    movel(p[x_c + 0.072285, y_c + -0.106434, z_c, rx, ry, rz], a, v)
    movel(p[x_c + 0.072329, y_c + -0.106475, z_c, rx, ry, rz], a, v)
    movel(p[x_c + 0.072376, y_c + -0.106518, z_c, rx, ry, rz], a, v)
    movel(p[x_c + 0.072426, y_c + -0.106564, z_c, rx, ry, rz], a, v)
    movel(p[x_c + 0.072479, y_c + -0.106612, z_c, rx, ry, rz], a, v)
    movel(p[x_c + 0.072535, y_c + -0.106663, z_c, rx, ry, rz], a, v)
    movel(p[x_c + 0.072593, y_c + -0.106716, z_c, rx, ry, rz], a, v)
    movel(p[x_c + 0.072654, y_c + -0.106772, z_c, rx, ry, rz], a, v)
    movel(p[x_c + 0.072718, y_c + -0.106830, z_c, rx, ry, rz], a, v)
    movel(p[x_c + 0.072785, y_c + -0.106890, z_c, rx, ry, rz], a, v)
    movel(p[x_c + 0.072855, y_c + -0.106954, z_c, rx, ry, rz], a, v)
    movel(p[x_c + 0.072855, y_c + -0.106954, z_c, rx, ry, rz], a, v)
    movel(p[x_c + 0.072959, y_c + -0.107049, z_c, rx, ry, rz], a, v)
    movel(p[x_c + 0.073072, y_c + -0.107153, z_c, rx, ry, rz], a, v)
    movel(p[x_c + 0.073193, y_c + -0.107267, z_c, rx, ry, rz], a, v)
    movel(p[x_c + 0.073322, y_c + -0.107389, z_c, rx, ry, rz], a, v)
    movel(p[x_c + 0.073459, y_c + -0.107519, z_c, rx, ry, rz], a, v)
    movel(p[x_c + 0.073603, y_c + -0.107657, z_c, rx, ry, rz], a, v)
    movel(p[x_c + 0.073754, y_c + -0.107802, z_c, rx, ry, rz], a, v)
    movel(p[x_c + 0.073910, y_c + -0.107953, z_c, rx, ry, rz], a, v)
    movel(p[x_c + 0.074072, y_c + -0.108111, z_c, rx, ry, rz], a, v)
    movel(p[x_c + 0.074240, y_c + -0.108275, z_c, rx, ry, rz], a, v)
    movel(p[x_c + 0.074412, y_c + -0.108443, z_c, rx, ry, rz], a, v)
    movel(p[x_c + 0.074589, y_c + -0.108617, z_c, rx, ry, rz], a, v)
    movel(p[x_c + 0.074769, y_c + -0.108795, z_c, rx, ry, rz], a, v)
    movel(p[x_c + 0.074953, y_c + -0.108977, z_c, rx, ry, rz], a, v)
    movel(p[x_c + 0.075139, y_c + -0.109162, z_c, rx, ry, rz], a, v)
    movel(p[x_c + 0.075329, y_c + -0.109350, z_c, rx, ry, rz], a, v)
    movel(p[x_c + 0.075520, y_c + -0.109541, z_c, rx, ry, rz], a, v)
    movel(p[x_c + 0.075712, y_c + -0.109734, z_c, rx, ry, rz], a, v)
    movel(p[x_c + 0.075906, y_c + -0.109928, z_c, rx, ry, rz], a, v)
    movel(p[x_c + 0.076100, y_c + -0.110123, z_c, rx, ry, rz], a, v)
    movel(p[x_c + 0.076295, y_c + -0.110319, z_c, rx, ry, rz], a, v)
    movel(p[x_c + 0.076489, y_c + -0.110515, z_c, rx, ry, rz], a, v)
    movel(p[x_c + 0.076683, y_c + -0.110711, z_c, rx, ry, rz], a, v)
    movel(p[x_c + 0.076875, y_c + -0.110906, z_c, rx, ry, rz], a, v)
    movel(p[x_c + 0.077065, y_c + -0.111099, z_c, rx, ry, rz], a, v)
    movel(p[x_c + 0.077254, y_c + -0.111291, z_c, rx, ry, rz], a, v)
    movel(p[x_c + 0.077440, y_c + -0.111481, z_c, rx, ry, rz], a, v)
    movel(p[x_c + 0.077622, y_c + -0.111668, z_c, rx, ry, rz], a, v)
    movel(p[x_c + 0.077802, y_c + -0.111852, z_c, rx, ry, rz], a, v)
    movel(p[x_c + 0.077977, y_c + -0.112032, z_c, rx, ry, rz], a, v)
    movel(p[x_c + 0.078148, y_c + -0.112209, z_c, rx, ry, rz], a, v)
    movel(p[x_c + 0.078314, y_c + -0.112380, z_c, rx, ry, rz], a, v)
    movel(p[x_c + 0.078474, y_c + -0.112547, z_c, rx, ry, rz], a, v)
    movel(p[x_c + 0.078629, y_c + -0.112708, z_c, rx, ry, rz], a, v)
    movel(p[x_c + 0.078778, y_c + -0.112864, z_c, rx, ry, rz], a, v)
    movel(p[x_c + 0.078919, y_c + -0.113013, z_c, rx, ry, rz], a, v)
    movel(p[x_c + 0.079054, y_c + -0.113155, z_c, rx, ry, rz], a, v)
    movel(p[x_c + 0.079181, y_c + -0.113290, z_c, rx, ry, rz], a, v)
    movel(p[x_c + 0.079300, y_c + -0.113417, z_c, rx, ry, rz], a, v)
    movel(p[x_c + 0.079410, y_c + -0.113535, z_c, rx, ry, rz], a, v)
    movel(p[x_c + 0.079511, y_c + -0.113645, z_c, rx, ry, rz], a, v)
    movel(p[x_c + 0.079603, y_c + -0.113746, z_c, rx, ry, rz], a, v)
    movel(p[x_c + 0.079685, y_c + -0.113837, z_c, rx, ry, rz], a, v)
    movel(p[x_c + 0.079756, y_c + -0.113918, z_c, rx, ry, rz], a, v)
    movel(p[x_c + 0.079817, y_c + -0.113989, z_c, rx, ry, rz], a, v)
    movel(p[x_c + 0.079866, y_c + -0.114048, z_c, rx, ry, rz], a, v)
    movel(p[x_c + 0.079904, y_c + -0.114096, z_c, rx, ry, rz], a, v)
    movel(p[x_c + 0.079929, y_c + -0.114132, z_c, rx, ry, rz], a, v)
    movel(p[x_c + 0.079941, y_c + -0.114155, z_c, rx, ry, rz], a, v)
    movel(p[x_c + 0.079941, y_c + -0.114155, z_c, rx, ry, rz], a, v)
    movel(p[x_c + 0.079943, y_c + -0.114162, z_c, rx, ry, rz], a, v)
    movel(p[x_c + 0.079943, y_c + -0.114167, z_c, rx, ry, rz], a, v)
    movel(p[x_c + 0.079941, y_c + -0.114171, z_c, rx, ry, rz], a, v)
    movel(p[x_c + 0.079937, y_c + -0.114173, z_c, rx, ry, rz], a, v)
    movel(p[x_c + 0.079932, y_c + -0.114175, z_c, rx, ry, rz], a, v)
    movel(p[x_c + 0.079924, y_c + -0.114175, z_c, rx, ry, rz], a, v)
    movel(p[x_c + 0.079916, y_c + -0.114173, z_c, rx, ry, rz], a, v)
    movel(p[x_c + 0.079905, y_c + -0.114171, z_c, rx, ry, rz], a, v)
    movel(p[x_c + 0.079892, y_c + -0.114167, z_c, rx, ry, rz], a, v)
    movel(p[x_c + 0.079878, y_c + -0.114162, z_c, rx, ry, rz], a, v)
    movel(p[x_c + 0.079863, y_c + -0.114155, z_c, rx, ry, rz], a, v)
    movel(p[x_c + 0.079846, y_c + -0.114148, z_c, rx, ry, rz], a, v)
    movel(p[x_c + 0.079827, y_c + -0.114139, z_c, rx, ry, rz], a, v)
    movel(p[x_c + 0.079807, y_c + -0.114129, z_c, rx, ry, rz], a, v)
    movel(p[x_c + 0.079785, y_c + -0.114119, z_c, rx, ry, rz], a, v)
    movel(p[x_c + 0.079762, y_c + -0.114106, z_c, rx, ry, rz], a, v)
    movel(p[x_c + 0.079737, y_c + -0.114093, z_c, rx, ry, rz], a, v)
    movel(p[x_c + 0.079711, y_c + -0.114079, z_c, rx, ry, rz], a, v)
    movel(p[x_c + 0.079684, y_c + -0.114064, z_c, rx, ry, rz], a, v)
    movel(p[x_c + 0.079655, y_c + -0.114047, z_c, rx, ry, rz], a, v)
    movel(p[x_c + 0.079625, y_c + -0.114030, z_c, rx, ry, rz], a, v)
    movel(p[x_c + 0.079593, y_c + -0.114012, z_c, rx, ry, rz], a, v)
    movel(p[x_c + 0.079561, y_c + -0.113992, z_c, rx, ry, rz], a, v)
    movel(p[x_c + 0.079527, y_c + -0.113972, z_c, rx, ry, rz], a, v)
    movel(p[x_c + 0.079492, y_c + -0.113950, z_c, rx, ry, rz], a, v)
    movel(p[x_c + 0.079455, y_c + -0.113928, z_c, rx, ry, rz], a, v)
    movel(p[x_c + 0.079418, y_c + -0.113905, z_c, rx, ry, rz], a, v)
    movel(p[x_c + 0.079379, y_c + -0.113881, z_c, rx, ry, rz], a, v)
    movel(p[x_c + 0.079340, y_c + -0.113856, z_c, rx, ry, rz], a, v)
    movel(p[x_c + 0.079299, y_c + -0.113830, z_c, rx, ry, rz], a, v)
    movel(p[x_c + 0.079257, y_c + -0.113803, z_c, rx, ry, rz], a, v)
    movel(p[x_c + 0.079214, y_c + -0.113775, z_c, rx, ry, rz], a, v)
    movel(p[x_c + 0.079171, y_c + -0.113747, z_c, rx, ry, rz], a, v)
    movel(p[x_c + 0.079126, y_c + -0.113718, z_c, rx, ry, rz], a, v)
    movel(p[x_c + 0.079080, y_c + -0.113688, z_c, rx, ry, rz], a, v)
    movel(p[x_c + 0.079034, y_c + -0.113657, z_c, rx, ry, rz], a, v)
    movel(p[x_c + 0.078987, y_c + -0.113625, z_c, rx, ry, rz], a, v)
    movel(p[x_c + 0.078938, y_c + -0.113593, z_c, rx, ry, rz], a, v)
    movel(p[x_c + 0.078889, y_c + -0.113560, z_c, rx, ry, rz], a, v)
    movel(p[x_c + 0.078840, y_c + -0.113526, z_c, rx, ry, rz], a, v)
    movel(p[x_c + 0.078789, y_c + -0.113492, z_c, rx, ry, rz], a, v)
    movel(p[x_c + 0.078738, y_c + -0.113457, z_c, rx, ry, rz], a, v)
    movel(p[x_c + 0.078686, y_c + -0.113421, z_c, rx, ry, rz], a, v)
    movel(p[x_c + 0.078633, y_c + -0.113384, z_c, rx, ry, rz], a, v)
    movel(p[x_c + 0.078580, y_c + -0.113347, z_c, rx, ry, rz], a, v)
    movel(p[x_c + 0.078526, y_c + -0.113310, z_c, rx, ry, rz], a, v)
    movel(p[x_c + 0.078472, y_c + -0.113272, z_c, rx, ry, rz], a, v)
    movel(p[x_c + 0.078417, y_c + -0.113233, z_c, rx, ry, rz], a, v)
    movel(p[x_c + 0.078361, y_c + -0.113193, z_c, rx, ry, rz], a, v)
    movel(p[x_c + 0.078361, y_c + -0.113193, z_c, rx, ry, rz], a, v)
    movel(p[x_c + 0.078071, y_c + -0.112987, z_c, rx, ry, rz], a, v)
    movel(p[x_c + 0.077789, y_c + -0.112787, z_c, rx, ry, rz], a, v)
    movel(p[x_c + 0.077513, y_c + -0.112592, z_c, rx, ry, rz], a, v)
    movel(p[x_c + 0.077245, y_c + -0.112401, z_c, rx, ry, rz], a, v)
    movel(p[x_c + 0.076983, y_c + -0.112216, z_c, rx, ry, rz], a, v)
    movel(p[x_c + 0.076728, y_c + -0.112036, z_c, rx, ry, rz], a, v)
    movel(p[x_c + 0.076480, y_c + -0.111861, z_c, rx, ry, rz], a, v)
    movel(p[x_c + 0.076238, y_c + -0.111690, z_c, rx, ry, rz], a, v)
    movel(p[x_c + 0.076002, y_c + -0.111524, z_c, rx, ry, rz], a, v)
    movel(p[x_c + 0.075773, y_c + -0.111363, z_c, rx, ry, rz], a, v)
    movel(p[x_c + 0.075549, y_c + -0.111206, z_c, rx, ry, rz], a, v)
    movel(p[x_c + 0.075331, y_c + -0.111054, z_c, rx, ry, rz], a, v)
    movel(p[x_c + 0.075119, y_c + -0.110905, z_c, rx, ry, rz], a, v)
    movel(p[x_c + 0.074913, y_c + -0.110761, z_c, rx, ry, rz], a, v)
    movel(p[x_c + 0.074711, y_c + -0.110621, z_c, rx, ry, rz], a, v)
    movel(p[x_c + 0.074515, y_c + -0.110485, z_c, rx, ry, rz], a, v)
    movel(p[x_c + 0.074324, y_c + -0.110353, z_c, rx, ry, rz], a, v)
    movel(p[x_c + 0.074138, y_c + -0.110224, z_c, rx, ry, rz], a, v)
    movel(p[x_c + 0.073957, y_c + -0.110099, z_c, rx, ry, rz], a, v)
    movel(p[x_c + 0.073780, y_c + -0.109978, z_c, rx, ry, rz], a, v)
    movel(p[x_c + 0.073608, y_c + -0.109860, z_c, rx, ry, rz], a, v)
    movel(p[x_c + 0.073440, y_c + -0.109745, z_c, rx, ry, rz], a, v)
    movel(p[x_c + 0.073276, y_c + -0.109634, z_c, rx, ry, rz], a, v)
    movel(p[x_c + 0.073117, y_c + -0.109526, z_c, rx, ry, rz], a, v)
    movel(p[x_c + 0.072961, y_c + -0.109420, z_c, rx, ry, rz], a, v)
    movel(p[x_c + 0.072809, y_c + -0.109318, z_c, rx, ry, rz], a, v)
    movel(p[x_c + 0.072660, y_c + -0.109219, z_c, rx, ry, rz], a, v)
    movel(p[x_c + 0.072515, y_c + -0.109122, z_c, rx, ry, rz], a, v)
    movel(p[x_c + 0.072373, y_c + -0.109028, z_c, rx, ry, rz], a, v)
    movel(p[x_c + 0.072234, y_c + -0.108936, z_c, rx, ry, rz], a, v)
    movel(p[x_c + 0.072098, y_c + -0.108847, z_c, rx, ry, rz], a, v)
    movel(p[x_c + 0.071965, y_c + -0.108760, z_c, rx, ry, rz], a, v)
    movel(p[x_c + 0.071834, y_c + -0.108675, z_c, rx, ry, rz], a, v)
    movel(p[x_c + 0.071706, y_c + -0.108593, z_c, rx, ry, rz], a, v)
    movel(p[x_c + 0.071581, y_c + -0.108512, z_c, rx, ry, rz], a, v)
    movel(p[x_c + 0.071457, y_c + -0.108433, z_c, rx, ry, rz], a, v)
    movel(p[x_c + 0.071336, y_c + -0.108357, z_c, rx, ry, rz], a, v)
    movel(p[x_c + 0.071216, y_c + -0.108281, z_c, rx, ry, rz], a, v)
    movel(p[x_c + 0.071099, y_c + -0.108208, z_c, rx, ry, rz], a, v)
    movel(p[x_c + 0.070983, y_c + -0.108136, z_c, rx, ry, rz], a, v)
    movel(p[x_c + 0.070868, y_c + -0.108065, z_c, rx, ry, rz], a, v)
    movel(p[x_c + 0.070755, y_c + -0.107996, z_c, rx, ry, rz], a, v)
    movel(p[x_c + 0.070642, y_c + -0.107928, z_c, rx, ry, rz], a, v)
    movel(p[x_c + 0.070531, y_c + -0.107861, z_c, rx, ry, rz], a, v)
    movel(p[x_c + 0.070421, y_c + -0.107795, z_c, rx, ry, rz], a, v)
    movel(p[x_c + 0.070311, y_c + -0.107729, z_c, rx, ry, rz], a, v)
    movel(p[x_c + 0.070202, y_c + -0.107665, z_c, rx, ry, rz], a, v)
    movel(p[x_c + 0.070093, y_c + -0.107601, z_c, rx, ry, rz], a, v)
    movel(p[x_c + 0.069984, y_c + -0.107538, z_c, rx, ry, rz], a, v)
    movel(p[x_c + 0.069984, y_c + -0.107538, z_c, rx, ry, rz], a, v)
    movel(p[x_c + 0.069919, y_c + -0.107500, z_c, rx, ry, rz], a, v)
    movel(p[x_c + 0.069853, y_c + -0.107462, z_c, rx, ry, rz], a, v)
    movel(p[x_c + 0.069787, y_c + -0.107423, z_c, rx, ry, rz], a, v)
    movel(p[x_c + 0.069721, y_c + -0.107385, z_c, rx, ry, rz], a, v)
    movel(p[x_c + 0.069654, y_c + -0.107346, z_c, rx, ry, rz], a, v)
    movel(p[x_c + 0.069588, y_c + -0.107308, z_c, rx, ry, rz], a, v)
    movel(p[x_c + 0.069522, y_c + -0.107269, z_c, rx, ry, rz], a, v)
    movel(p[x_c + 0.069456, y_c + -0.107230, z_c, rx, ry, rz], a, v)
    movel(p[x_c + 0.069391, y_c + -0.107192, z_c, rx, ry, rz], a, v)
    movel(p[x_c + 0.069325, y_c + -0.107153, z_c, rx, ry, rz], a, v)
    movel(p[x_c + 0.069260, y_c + -0.107115, z_c, rx, ry, rz], a, v)
    movel(p[x_c + 0.069195, y_c + -0.107077, z_c, rx, ry, rz], a, v)
    movel(p[x_c + 0.069130, y_c + -0.107039, z_c, rx, ry, rz], a, v)
    movel(p[x_c + 0.069066, y_c + -0.107001, z_c, rx, ry, rz], a, v)
    movel(p[x_c + 0.069002, y_c + -0.106963, z_c, rx, ry, rz], a, v)
    movel(p[x_c + 0.068939, y_c + -0.106926, z_c, rx, ry, rz], a, v)
    movel(p[x_c + 0.068876, y_c + -0.106889, z_c, rx, ry, rz], a, v)
    movel(p[x_c + 0.068814, y_c + -0.106852, z_c, rx, ry, rz], a, v)
    movel(p[x_c + 0.068752, y_c + -0.106815, z_c, rx, ry, rz], a, v)
    movel(p[x_c + 0.068691, y_c + -0.106779, z_c, rx, ry, rz], a, v)
    movel(p[x_c + 0.068631, y_c + -0.106743, z_c, rx, ry, rz], a, v)
    movel(p[x_c + 0.068572, y_c + -0.106708, z_c, rx, ry, rz], a, v)
    movel(p[x_c + 0.068513, y_c + -0.106673, z_c, rx, ry, rz], a, v)
    movel(p[x_c + 0.068455, y_c + -0.106639, z_c, rx, ry, rz], a, v)
    movel(p[x_c + 0.068398, y_c + -0.106605, z_c, rx, ry, rz], a, v)
    movel(p[x_c + 0.068342, y_c + -0.106571, z_c, rx, ry, rz], a, v)
    movel(p[x_c + 0.068287, y_c + -0.106538, z_c, rx, ry, rz], a, v)
    movel(p[x_c + 0.068233, y_c + -0.106506, z_c, rx, ry, rz], a, v)
    movel(p[x_c + 0.068181, y_c + -0.106474, z_c, rx, ry, rz], a, v)
    movel(p[x_c + 0.068129, y_c + -0.106443, z_c, rx, ry, rz], a, v)
    movel(p[x_c + 0.068078, y_c + -0.106412, z_c, rx, ry, rz], a, v)
    movel(p[x_c + 0.068029, y_c + -0.106382, z_c, rx, ry, rz], a, v)
    movel(p[x_c + 0.067981, y_c + -0.106353, z_c, rx, ry, rz], a, v)
    movel(p[x_c + 0.067934, y_c + -0.106325, z_c, rx, ry, rz], a, v)
    movel(p[x_c + 0.067889, y_c + -0.106297, z_c, rx, ry, rz], a, v)
    movel(p[x_c + 0.067844, y_c + -0.106270, z_c, rx, ry, rz], a, v)
    movel(p[x_c + 0.067802, y_c + -0.106244, z_c, rx, ry, rz], a, v)
    movel(p[x_c + 0.067761, y_c + -0.106219, z_c, rx, ry, rz], a, v)
    movel(p[x_c + 0.067721, y_c + -0.106195, z_c, rx, ry, rz], a, v)
    movel(p[x_c + 0.067683, y_c + -0.106171, z_c, rx, ry, rz], a, v)
    movel(p[x_c + 0.067647, y_c + -0.106149, z_c, rx, ry, rz], a, v)
    movel(p[x_c + 0.067612, y_c + -0.106127, z_c, rx, ry, rz], a, v)
    movel(p[x_c + 0.067579, y_c + -0.106107, z_c, rx, ry, rz], a, v)
    movel(p[x_c + 0.067548, y_c + -0.106087, z_c, rx, ry, rz], a, v)
    movel(p[x_c + 0.067519, y_c + -0.106069, z_c, rx, ry, rz], a, v)
    movel(p[x_c + 0.067491, y_c + -0.106051, z_c, rx, ry, rz], a, v)
    movel(p[x_c + 0.067466, y_c + -0.106035, z_c, rx, ry, rz], a, v)
    movel(p[x_c + 0.067442, y_c + -0.106020, z_c, rx, ry, rz], a, v)
    movel(p[x_c + 0.067420, y_c + -0.106006, z_c, rx, ry, rz], a, v)
    movel(p[x_c + 0.067420, y_c + -0.106006, z_c, rx, ry, rz], a, v)
    movel(p[x_c + 0.067361, y_c + -0.105967, z_c, rx, ry, rz], a, v)
    movel(p[x_c + 0.067304, y_c + -0.105930, z_c, rx, ry, rz], a, v)
    movel(p[x_c + 0.067251, y_c + -0.105897, z_c, rx, ry, rz], a, v)
    movel(p[x_c + 0.067201, y_c + -0.105865, z_c, rx, ry, rz], a, v)
    movel(p[x_c + 0.067154, y_c + -0.105837, z_c, rx, ry, rz], a, v)
    movel(p[x_c + 0.067110, y_c + -0.105810, z_c, rx, ry, rz], a, v)
    movel(p[x_c + 0.067070, y_c + -0.105787, z_c, rx, ry, rz], a, v)
    movel(p[x_c + 0.067032, y_c + -0.105765, z_c, rx, ry, rz], a, v)
    movel(p[x_c + 0.066998, y_c + -0.105746, z_c, rx, ry, rz], a, v)
    movel(p[x_c + 0.066966, y_c + -0.105729, z_c, rx, ry, rz], a, v)
    movel(p[x_c + 0.066938, y_c + -0.105715, z_c, rx, ry, rz], a, v)
    movel(p[x_c + 0.066912, y_c + -0.105703, z_c, rx, ry, rz], a, v)
    movel(p[x_c + 0.066890, y_c + -0.105693, z_c, rx, ry, rz], a, v)
    movel(p[x_c + 0.066870, y_c + -0.105685, z_c, rx, ry, rz], a, v)
    movel(p[x_c + 0.066853, y_c + -0.105679, z_c, rx, ry, rz], a, v)
    movel(p[x_c + 0.066839, y_c + -0.105676, z_c, rx, ry, rz], a, v)
    movel(p[x_c + 0.066828, y_c + -0.105674, z_c, rx, ry, rz], a, v)
    movel(p[x_c + 0.066820, y_c + -0.105675, z_c, rx, ry, rz], a, v)
    movel(p[x_c + 0.066815, y_c + -0.105677, z_c, rx, ry, rz], a, v)
    movel(p[x_c + 0.066812, y_c + -0.105682, z_c, rx, ry, rz], a, v)
    movel(p[x_c + 0.066812, y_c + -0.105689, z_c, rx, ry, rz], a, v)
    movel(p[x_c + 0.066815, y_c + -0.105697, z_c, rx, ry, rz], a, v)
    movel(p[x_c + 0.066821, y_c + -0.105708, z_c, rx, ry, rz], a, v)
    movel(p[x_c + 0.066829, y_c + -0.105720, z_c, rx, ry, rz], a, v)
    movel(p[x_c + 0.066840, y_c + -0.105734, z_c, rx, ry, rz], a, v)
    movel(p[x_c + 0.066853, y_c + -0.105750, z_c, rx, ry, rz], a, v)
    movel(p[x_c + 0.066869, y_c + -0.105768, z_c, rx, ry, rz], a, v)
    movel(p[x_c + 0.066888, y_c + -0.105787, z_c, rx, ry, rz], a, v)
    movel(p[x_c + 0.066909, y_c + -0.105808, z_c, rx, ry, rz], a, v)
    movel(p[x_c + 0.066933, y_c + -0.105831, z_c, rx, ry, rz], a, v)
    movel(p[x_c + 0.066959, y_c + -0.105855, z_c, rx, ry, rz], a, v)
    movel(p[x_c + 0.066988, y_c + -0.105881, z_c, rx, ry, rz], a, v)
    movel(p[x_c + 0.067019, y_c + -0.105909, z_c, rx, ry, rz], a, v)
    movel(p[x_c + 0.067053, y_c + -0.105938, z_c, rx, ry, rz], a, v)
    movel(p[x_c + 0.067089, y_c + -0.105969, z_c, rx, ry, rz], a, v)
    movel(p[x_c + 0.067127, y_c + -0.106001, z_c, rx, ry, rz], a, v)
    movel(p[x_c + 0.067168, y_c + -0.106034, z_c, rx, ry, rz], a, v)
    movel(p[x_c + 0.067211, y_c + -0.106069, z_c, rx, ry, rz], a, v)
    movel(p[x_c + 0.067256, y_c + -0.106106, z_c, rx, ry, rz], a, v)
    movel(p[x_c + 0.067304, y_c + -0.106143, z_c, rx, ry, rz], a, v)
    movel(p[x_c + 0.067353, y_c + -0.106182, z_c, rx, ry, rz], a, v)
    movel(p[x_c + 0.067405, y_c + -0.106223, z_c, rx, ry, rz], a, v)
    movel(p[x_c + 0.067460, y_c + -0.106264, z_c, rx, ry, rz], a, v)
    movel(p[x_c + 0.067516, y_c + -0.106307, z_c, rx, ry, rz], a, v)
    movel(p[x_c + 0.067575, y_c + -0.106351, z_c, rx, ry, rz], a, v)
    movel(p[x_c + 0.067635, y_c + -0.106396, z_c, rx, ry, rz], a, v)
    movel(p[x_c + 0.067698, y_c + -0.106442, z_c, rx, ry, rz], a, v)
    movel(p[x_c + 0.067763, y_c + -0.106489, z_c, rx, ry, rz], a, v)
    movel(p[x_c + 0.067830, y_c + -0.106537, z_c, rx, ry, rz], a, v)
    movel(p[x_c + 0.067830, y_c + -0.106537, z_c, rx, ry, rz], a, v)
    movel(p[x_c + 0.067865, y_c + -0.106563, z_c, rx, ry, rz], a, v)
    movel(p[x_c + 0.067903, y_c + -0.106591, z_c, rx, ry, rz], a, v)
    movel(p[x_c + 0.067944, y_c + -0.106620, z_c, rx, ry, rz], a, v)
    movel(p[x_c + 0.067986, y_c + -0.106652, z_c, rx, ry, rz], a, v)
    movel(p[x_c + 0.068031, y_c + -0.106685, z_c, rx, ry, rz], a, v)
    movel(p[x_c + 0.068077, y_c + -0.106721, z_c, rx, ry, rz], a, v)
    movel(p[x_c + 0.068126, y_c + -0.106758, z_c, rx, ry, rz], a, v)
    movel(p[x_c + 0.068177, y_c + -0.106797, z_c, rx, ry, rz], a, v)
    movel(p[x_c + 0.068229, y_c + -0.106837, z_c, rx, ry, rz], a, v)
    movel(p[x_c + 0.068284, y_c + -0.106879, z_c, rx, ry, rz], a, v)
    movel(p[x_c + 0.068340, y_c + -0.106922, z_c, rx, ry, rz], a, v)
    movel(p[x_c + 0.068398, y_c + -0.106968, z_c, rx, ry, rz], a, v)
    movel(p[x_c + 0.068458, y_c + -0.107014, z_c, rx, ry, rz], a, v)
    movel(p[x_c + 0.068519, y_c + -0.107062, z_c, rx, ry, rz], a, v)
    movel(p[x_c + 0.068582, y_c + -0.107111, z_c, rx, ry, rz], a, v)
    movel(p[x_c + 0.068646, y_c + -0.107162, z_c, rx, ry, rz], a, v)
    movel(p[x_c + 0.068712, y_c + -0.107214, z_c, rx, ry, rz], a, v)
    movel(p[x_c + 0.068779, y_c + -0.107267, z_c, rx, ry, rz], a, v)
    movel(p[x_c + 0.068847, y_c + -0.107321, z_c, rx, ry, rz], a, v)
    movel(p[x_c + 0.068917, y_c + -0.107377, z_c, rx, ry, rz], a, v)
    movel(p[x_c + 0.068988, y_c + -0.107433, z_c, rx, ry, rz], a, v)
    movel(p[x_c + 0.069060, y_c + -0.107491, z_c, rx, ry, rz], a, v)
    movel(p[x_c + 0.069133, y_c + -0.107549, z_c, rx, ry, rz], a, v)
    movel(p[x_c + 0.069207, y_c + -0.107609, z_c, rx, ry, rz], a, v)
    movel(p[x_c + 0.069281, y_c + -0.107669, z_c, rx, ry, rz], a, v)
    movel(p[x_c + 0.069357, y_c + -0.107730, z_c, rx, ry, rz], a, v)
    movel(p[x_c + 0.069434, y_c + -0.107792, z_c, rx, ry, rz], a, v)
    movel(p[x_c + 0.069511, y_c + -0.107855, z_c, rx, ry, rz], a, v)
    movel(p[x_c + 0.069589, y_c + -0.107918, z_c, rx, ry, rz], a, v)
    movel(p[x_c + 0.069668, y_c + -0.107982, z_c, rx, ry, rz], a, v)
    movel(p[x_c + 0.069747, y_c + -0.108047, z_c, rx, ry, rz], a, v)
    movel(p[x_c + 0.069827, y_c + -0.108112, z_c, rx, ry, rz], a, v)
    movel(p[x_c + 0.069908, y_c + -0.108178, z_c, rx, ry, rz], a, v)
    movel(p[x_c + 0.069988, y_c + -0.108244, z_c, rx, ry, rz], a, v)
    movel(p[x_c + 0.070069, y_c + -0.108310, z_c, rx, ry, rz], a, v)
    movel(p[x_c + 0.070151, y_c + -0.108377, z_c, rx, ry, rz], a, v)
    movel(p[x_c + 0.070232, y_c + -0.108444, z_c, rx, ry, rz], a, v)
    movel(p[x_c + 0.070314, y_c + -0.108511, z_c, rx, ry, rz], a, v)
    movel(p[x_c + 0.070396, y_c + -0.108579, z_c, rx, ry, rz], a, v)
    movel(p[x_c + 0.070477, y_c + -0.108647, z_c, rx, ry, rz], a, v)
    movel(p[x_c + 0.070559, y_c + -0.108714, z_c, rx, ry, rz], a, v)
    movel(p[x_c + 0.070641, y_c + -0.108782, z_c, rx, ry, rz], a, v)
    movel(p[x_c + 0.070723, y_c + -0.108850, z_c, rx, ry, rz], a, v)
    movel(p[x_c + 0.070804, y_c + -0.108918, z_c, rx, ry, rz], a, v)
    movel(p[x_c + 0.070885, y_c + -0.108986, z_c, rx, ry, rz], a, v)
    movel(p[x_c + 0.070966, y_c + -0.109053, z_c, rx, ry, rz], a, v)
    movel(p[x_c + 0.071046, y_c + -0.109121, z_c, rx, ry, rz], a, v)
    movel(p[x_c + 0.071126, y_c + -0.109188, z_c, rx, ry, rz], a, v)
    movel(p[x_c + 0.071206, y_c + -0.109255, z_c, rx, ry, rz], a, v)
    movel(p[x_c + 0.071206, y_c + -0.109255, z_c, rx, ry, rz], a, v)
    movel(p[x_c + 0.071285, y_c + -0.109322, z_c, rx, ry, rz], a, v)
    movel(p[x_c + 0.071364, y_c + -0.109389, z_c, rx, ry, rz], a, v)
    movel(p[x_c + 0.071443, y_c + -0.109455, z_c, rx, ry, rz], a, v)
    movel(p[x_c + 0.071523, y_c + -0.109522, z_c, rx, ry, rz], a, v)
    movel(p[x_c + 0.071602, y_c + -0.109588, z_c, rx, ry, rz], a, v)
    movel(p[x_c + 0.071680, y_c + -0.109654, z_c, rx, ry, rz], a, v)
    movel(p[x_c + 0.071759, y_c + -0.109720, z_c, rx, ry, rz], a, v)
    movel(p[x_c + 0.071837, y_c + -0.109786, z_c, rx, ry, rz], a, v)
    movel(p[x_c + 0.071915, y_c + -0.109852, z_c, rx, ry, rz], a, v)
    movel(p[x_c + 0.071993, y_c + -0.109917, z_c, rx, ry, rz], a, v)
    movel(p[x_c + 0.072070, y_c + -0.109981, z_c, rx, ry, rz], a, v)
    movel(p[x_c + 0.072146, y_c + -0.110045, z_c, rx, ry, rz], a, v)
    movel(p[x_c + 0.072222, y_c + -0.110109, z_c, rx, ry, rz], a, v)
    movel(p[x_c + 0.072298, y_c + -0.110172, z_c, rx, ry, rz], a, v)
    movel(p[x_c + 0.072372, y_c + -0.110234, z_c, rx, ry, rz], a, v)
    movel(p[x_c + 0.072446, y_c + -0.110296, z_c, rx, ry, rz], a, v)
    movel(p[x_c + 0.072520, y_c + -0.110358, z_c, rx, ry, rz], a, v)
    movel(p[x_c + 0.072592, y_c + -0.110418, z_c, rx, ry, rz], a, v)
    movel(p[x_c + 0.072664, y_c + -0.110478, z_c, rx, ry, rz], a, v)
    movel(p[x_c + 0.072734, y_c + -0.110537, z_c, rx, ry, rz], a, v)
    movel(p[x_c + 0.072804, y_c + -0.110595, z_c, rx, ry, rz], a, v)
    movel(p[x_c + 0.072873, y_c + -0.110652, z_c, rx, ry, rz], a, v)
    movel(p[x_c + 0.072940, y_c + -0.110708, z_c, rx, ry, rz], a, v)
    movel(p[x_c + 0.073006, y_c + -0.110763, z_c, rx, ry, rz], a, v)
    movel(p[x_c + 0.073072, y_c + -0.110817, z_c, rx, ry, rz], a, v)
    movel(p[x_c + 0.073136, y_c + -0.110871, z_c, rx, ry, rz], a, v)
    movel(p[x_c + 0.073198, y_c + -0.110923, z_c, rx, ry, rz], a, v)
    movel(p[x_c + 0.073260, y_c + -0.110973, z_c, rx, ry, rz], a, v)
    movel(p[x_c + 0.073320, y_c + -0.111023, z_c, rx, ry, rz], a, v)
    movel(p[x_c + 0.073378, y_c + -0.111071, z_c, rx, ry, rz], a, v)
    movel(p[x_c + 0.073435, y_c + -0.111119, z_c, rx, ry, rz], a, v)
    movel(p[x_c + 0.073491, y_c + -0.111164, z_c, rx, ry, rz], a, v)
    movel(p[x_c + 0.073544, y_c + -0.111209, z_c, rx, ry, rz], a, v)
    movel(p[x_c + 0.073597, y_c + -0.111252, z_c, rx, ry, rz], a, v)
    movel(p[x_c + 0.073647, y_c + -0.111293, z_c, rx, ry, rz], a, v)
    movel(p[x_c + 0.073696, y_c + -0.111333, z_c, rx, ry, rz], a, v)
    movel(p[x_c + 0.073743, y_c + -0.111372, z_c, rx, ry, rz], a, v)
    movel(p[x_c + 0.073788, y_c + -0.111409, z_c, rx, ry, rz], a, v)
    movel(p[x_c + 0.073831, y_c + -0.111444, z_c, rx, ry, rz], a, v)
    movel(p[x_c + 0.073872, y_c + -0.111478, z_c, rx, ry, rz], a, v)
    movel(p[x_c + 0.073911, y_c + -0.111510, z_c, rx, ry, rz], a, v)
    movel(p[x_c + 0.073948, y_c + -0.111540, z_c, rx, ry, rz], a, v)
    movel(p[x_c + 0.073983, y_c + -0.111568, z_c, rx, ry, rz], a, v)
    movel(p[x_c + 0.074015, y_c + -0.111595, z_c, rx, ry, rz], a, v)
    movel(p[x_c + 0.074046, y_c + -0.111619, z_c, rx, ry, rz], a, v)
    movel(p[x_c + 0.074074, y_c + -0.111642, z_c, rx, ry, rz], a, v)
    movel(p[x_c + 0.074100, y_c + -0.111662, z_c, rx, ry, rz], a, v)
    movel(p[x_c + 0.074123, y_c + -0.111681, z_c, rx, ry, rz], a, v)
    movel(p[x_c + 0.074144, y_c + -0.111698, z_c, rx, ry, rz], a, v)
    movel(p[x_c + 0.074144, y_c + -0.111698, z_c, rx, ry, rz], a, v)
    movel(p[x_c + 0.074200, y_c + -0.111741, z_c, rx, ry, rz], a, v)
    movel(p[x_c + 0.074251, y_c + -0.111782, z_c, rx, ry, rz], a, v)
    movel(p[x_c + 0.074297, y_c + -0.111819, z_c, rx, ry, rz], a, v)
    movel(p[x_c + 0.074339, y_c + -0.111853, z_c, rx, ry, rz], a, v)
    movel(p[x_c + 0.074377, y_c + -0.111884, z_c, rx, ry, rz], a, v)
    movel(p[x_c + 0.074409, y_c + -0.111912, z_c, rx, ry, rz], a, v)
    movel(p[x_c + 0.074438, y_c + -0.111937, z_c, rx, ry, rz], a, v)
    movel(p[x_c + 0.074461, y_c + -0.111958, z_c, rx, ry, rz], a, v)
    movel(p[x_c + 0.074480, y_c + -0.111976, z_c, rx, ry, rz], a, v)
    movel(p[x_c + 0.074494, y_c + -0.111991, z_c, rx, ry, rz], a, v)
    movel(p[x_c + 0.074504, y_c + -0.112003, z_c, rx, ry, rz], a, v)
    movel(p[x_c + 0.074508, y_c + -0.112011, z_c, rx, ry, rz], a, v)
    movel(p[x_c + 0.074508, y_c + -0.112016, z_c, rx, ry, rz], a, v)
    movel(p[x_c + 0.074504, y_c + -0.112018, z_c, rx, ry, rz], a, v)
    movel(p[x_c + 0.074494, y_c + -0.112016, z_c, rx, ry, rz], a, v)
    movel(p[x_c + 0.074480, y_c + -0.112011, z_c, rx, ry, rz], a, v)
    movel(p[x_c + 0.074461, y_c + -0.112003, z_c, rx, ry, rz], a, v)
    movel(p[x_c + 0.074437, y_c + -0.111991, z_c, rx, ry, rz], a, v)
    movel(p[x_c + 0.074408, y_c + -0.111976, z_c, rx, ry, rz], a, v)
    movel(p[x_c + 0.074374, y_c + -0.111958, z_c, rx, ry, rz], a, v)
    movel(p[x_c + 0.074335, y_c + -0.111936, z_c, rx, ry, rz], a, v)
    movel(p[x_c + 0.074291, y_c + -0.111911, z_c, rx, ry, rz], a, v)
    movel(p[x_c + 0.074242, y_c + -0.111882, z_c, rx, ry, rz], a, v)
    movel(p[x_c + 0.074189, y_c + -0.111850, z_c, rx, ry, rz], a, v)
    movel(p[x_c + 0.074130, y_c + -0.111815, z_c, rx, ry, rz], a, v)
    movel(p[x_c + 0.074066, y_c + -0.111775, z_c, rx, ry, rz], a, v)
    movel(p[x_c + 0.073997, y_c + -0.111733, z_c, rx, ry, rz], a, v)
    movel(p[x_c + 0.073923, y_c + -0.111687, z_c, rx, ry, rz], a, v)
    movel(p[x_c + 0.073844, y_c + -0.111637, z_c, rx, ry, rz], a, v)
    movel(p[x_c + 0.073760, y_c + -0.111584, z_c, rx, ry, rz], a, v)
    movel(p[x_c + 0.073670, y_c + -0.111528, z_c, rx, ry, rz], a, v)
    movel(p[x_c + 0.073576, y_c + -0.111467, z_c, rx, ry, rz], a, v)
    movel(p[x_c + 0.073476, y_c + -0.111403, z_c, rx, ry, rz], a, v)
    movel(p[x_c + 0.073371, y_c + -0.111336, z_c, rx, ry, rz], a, v)
    movel(p[x_c + 0.073260, y_c + -0.111265, z_c, rx, ry, rz], a, v)
    movel(p[x_c + 0.073145, y_c + -0.111190, z_c, rx, ry, rz], a, v)
    movel(p[x_c + 0.073024, y_c + -0.111112, z_c, rx, ry, rz], a, v)
    movel(p[x_c + 0.072898, y_c + -0.111030, z_c, rx, ry, rz], a, v)
    movel(p[x_c + 0.072766, y_c + -0.110945, z_c, rx, ry, rz], a, v)
    movel(p[x_c + 0.072629, y_c + -0.110855, z_c, rx, ry, rz], a, v)
    movel(p[x_c + 0.072486, y_c + -0.110763, z_c, rx, ry, rz], a, v)
    movel(p[x_c + 0.072339, y_c + -0.110666, z_c, rx, ry, rz], a, v)
    movel(p[x_c + 0.072185, y_c + -0.110566, z_c, rx, ry, rz], a, v)
    movel(p[x_c + 0.072027, y_c + -0.110461, z_c, rx, ry, rz], a, v)
    movel(p[x_c + 0.071862, y_c + -0.110354, z_c, rx, ry, rz], a, v)
    movel(p[x_c + 0.071693, y_c + -0.110242, z_c, rx, ry, rz], a, v)
    movel(p[x_c + 0.071517, y_c + -0.110127, z_c, rx, ry, rz], a, v)
    movel(p[x_c + 0.071336, y_c + -0.110008, z_c, rx, ry, rz], a, v)
    movel(p[x_c + 0.071150, y_c + -0.109885, z_c, rx, ry, rz], a, v)
    movel(p[x_c + 0.071150, y_c + -0.109885, z_c, rx, ry, rz], a, v)
    movel(p[x_c + 0.071052, y_c + -0.109820, z_c, rx, ry, rz], a, v)
    movel(p[x_c + 0.070953, y_c + -0.109755, z_c, rx, ry, rz], a, v)
    movel(p[x_c + 0.070853, y_c + -0.109689, z_c, rx, ry, rz], a, v)
    movel(p[x_c + 0.070753, y_c + -0.109623, z_c, rx, ry, rz], a, v)
    movel(p[x_c + 0.070651, y_c + -0.109556, z_c, rx, ry, rz], a, v)
    movel(p[x_c + 0.070549, y_c + -0.109489, z_c, rx, ry, rz], a, v)
    movel(p[x_c + 0.070446, y_c + -0.109422, z_c, rx, ry, rz], a, v)
    movel(p[x_c + 0.070343, y_c + -0.109355, z_c, rx, ry, rz], a, v)
    movel(p[x_c + 0.070239, y_c + -0.109287, z_c, rx, ry, rz], a, v)
    movel(p[x_c + 0.070135, y_c + -0.109219, z_c, rx, ry, rz], a, v)
    movel(p[x_c + 0.070030, y_c + -0.109151, z_c, rx, ry, rz], a, v)
    movel(p[x_c + 0.069926, y_c + -0.109082, z_c, rx, ry, rz], a, v)
    movel(p[x_c + 0.069821, y_c + -0.109014, z_c, rx, ry, rz], a, v)
    movel(p[x_c + 0.069716, y_c + -0.108946, z_c, rx, ry, rz], a, v)
    movel(p[x_c + 0.069611, y_c + -0.108878, z_c, rx, ry, rz], a, v)
    movel(p[x_c + 0.069507, y_c + -0.108810, z_c, rx, ry, rz], a, v)
    movel(p[x_c + 0.069402, y_c + -0.108742, z_c, rx, ry, rz], a, v)
    movel(p[x_c + 0.069298, y_c + -0.108675, z_c, rx, ry, rz], a, v)
    movel(p[x_c + 0.069194, y_c + -0.108607, z_c, rx, ry, rz], a, v)
    movel(p[x_c + 0.069091, y_c + -0.108541, z_c, rx, ry, rz], a, v)
    movel(p[x_c + 0.068988, y_c + -0.108474, z_c, rx, ry, rz], a, v)
    movel(p[x_c + 0.068886, y_c + -0.108408, z_c, rx, ry, rz], a, v)
    movel(p[x_c + 0.068784, y_c + -0.108342, z_c, rx, ry, rz], a, v)
    movel(p[x_c + 0.068683, y_c + -0.108277, z_c, rx, ry, rz], a, v)
    movel(p[x_c + 0.068583, y_c + -0.108213, z_c, rx, ry, rz], a, v)
    movel(p[x_c + 0.068484, y_c + -0.108149, z_c, rx, ry, rz], a, v)
    movel(p[x_c + 0.068386, y_c + -0.108086, z_c, rx, ry, rz], a, v)
    movel(p[x_c + 0.068289, y_c + -0.108024, z_c, rx, ry, rz], a, v)
    movel(p[x_c + 0.068194, y_c + -0.107962, z_c, rx, ry, rz], a, v)
    movel(p[x_c + 0.068099, y_c + -0.107902, z_c, rx, ry, rz], a, v)
    movel(p[x_c + 0.068006, y_c + -0.107842, z_c, rx, ry, rz], a, v)
    movel(p[x_c + 0.067914, y_c + -0.107783, z_c, rx, ry, rz], a, v)
    movel(p[x_c + 0.067823, y_c + -0.107726, z_c, rx, ry, rz], a, v)
    movel(p[x_c + 0.067735, y_c + -0.107669, z_c, rx, ry, rz], a, v)
    movel(p[x_c + 0.067647, y_c + -0.107614, z_c, rx, ry, rz], a, v)
    movel(p[x_c + 0.067562, y_c + -0.107559, z_c, rx, ry, rz], a, v)
    movel(p[x_c + 0.067478, y_c + -0.107506, z_c, rx, ry, rz], a, v)
    movel(p[x_c + 0.067397, y_c + -0.107454, z_c, rx, ry, rz], a, v)
    movel(p[x_c + 0.067317, y_c + -0.107404, z_c, rx, ry, rz], a, v)
    movel(p[x_c + 0.067239, y_c + -0.107354, z_c, rx, ry, rz], a, v)
    movel(p[x_c + 0.067163, y_c + -0.107307, z_c, rx, ry, rz], a, v)
    movel(p[x_c + 0.067090, y_c + -0.107260, z_c, rx, ry, rz], a, v)
    movel(p[x_c + 0.067019, y_c + -0.107216, z_c, rx, ry, rz], a, v)
    movel(p[x_c + 0.066950, y_c + -0.107173, z_c, rx, ry, rz], a, v)
    movel(p[x_c + 0.066884, y_c + -0.107131, z_c, rx, ry, rz], a, v)
    movel(p[x_c + 0.066820, y_c + -0.107091, z_c, rx, ry, rz], a, v)
    movel(p[x_c + 0.066759, y_c + -0.107053, z_c, rx, ry, rz], a, v)
    movel(p[x_c + 0.066700, y_c + -0.107017, z_c, rx, ry, rz], a, v)
    movel(p[x_c + 0.066645, y_c + -0.106983, z_c, rx, ry, rz], a, v)
    movel(p[x_c + 0.066645, y_c + -0.106983, z_c, rx, ry, rz], a, v)
    movel(p[x_c + 0.066590, y_c + -0.106949, z_c, rx, ry, rz], a, v)
    movel(p[x_c + 0.066533, y_c + -0.106914, z_c, rx, ry, rz], a, v)
    movel(p[x_c + 0.066476, y_c + -0.106878, z_c, rx, ry, rz], a, v)
    movel(p[x_c + 0.066417, y_c + -0.106842, z_c, rx, ry, rz], a, v)
    movel(p[x_c + 0.066357, y_c + -0.106805, z_c, rx, ry, rz], a, v)
    movel(p[x_c + 0.066295, y_c + -0.106767, z_c, rx, ry, rz], a, v)
    movel(p[x_c + 0.066233, y_c + -0.106728, z_c, rx, ry, rz], a, v)
    movel(p[x_c + 0.066170, y_c + -0.106689, z_c, rx, ry, rz], a, v)
    movel(p[x_c + 0.066105, y_c + -0.106649, z_c, rx, ry, rz], a, v)
    movel(p[x_c + 0.066040, y_c + -0.106608, z_c, rx, ry, rz], a, v)
    movel(p[x_c + 0.065974, y_c + -0.106567, z_c, rx, ry, rz], a, v)
    movel(p[x_c + 0.065907, y_c + -0.106525, z_c, rx, ry, rz], a, v)
    movel(p[x_c + 0.065840, y_c + -0.106483, z_c, rx, ry, rz], a, v)
    movel(p[x_c + 0.065772, y_c + -0.106440, z_c, rx, ry, rz], a, v)
    movel(p[x_c + 0.065703, y_c + -0.106397, z_c, rx, ry, rz], a, v)
    movel(p[x_c + 0.065633, y_c + -0.106354, z_c, rx, ry, rz], a, v)
    movel(p[x_c + 0.065563, y_c + -0.106310, z_c, rx, ry, rz], a, v)
    movel(p[x_c + 0.065493, y_c + -0.106266, z_c, rx, ry, rz], a, v)
    movel(p[x_c + 0.065422, y_c + -0.106222, z_c, rx, ry, rz], a, v)
    movel(p[x_c + 0.065351, y_c + -0.106177, z_c, rx, ry, rz], a, v)
    movel(p[x_c + 0.065280, y_c + -0.106132, z_c, rx, ry, rz], a, v)
    movel(p[x_c + 0.065209, y_c + -0.106087, z_c, rx, ry, rz], a, v)
    movel(p[x_c + 0.065137, y_c + -0.106042, z_c, rx, ry, rz], a, v)
    movel(p[x_c + 0.065065, y_c + -0.105997, z_c, rx, ry, rz], a, v)
    movel(p[x_c + 0.064993, y_c + -0.105952, z_c, rx, ry, rz], a, v)
    movel(p[x_c + 0.064922, y_c + -0.105907, z_c, rx, ry, rz], a, v)
    movel(p[x_c + 0.064850, y_c + -0.105862, z_c, rx, ry, rz], a, v)
    movel(p[x_c + 0.064778, y_c + -0.105816, z_c, rx, ry, rz], a, v)
    movel(p[x_c + 0.064707, y_c + -0.105771, z_c, rx, ry, rz], a, v)
    movel(p[x_c + 0.064636, y_c + -0.105726, z_c, rx, ry, rz], a, v)
    movel(p[x_c + 0.064565, y_c + -0.105682, z_c, rx, ry, rz], a, v)
    movel(p[x_c + 0.064495, y_c + -0.105637, z_c, rx, ry, rz], a, v)
    movel(p[x_c + 0.064425, y_c + -0.105593, z_c, rx, ry, rz], a, v)
    movel(p[x_c + 0.064355, y_c + -0.105549, z_c, rx, ry, rz], a, v)
    movel(p[x_c + 0.064286, y_c + -0.105505, z_c, rx, ry, rz], a, v)
    movel(p[x_c + 0.064218, y_c + -0.105462, z_c, rx, ry, rz], a, v)
    movel(p[x_c + 0.064150, y_c + -0.105419, z_c, rx, ry, rz], a, v)
    movel(p[x_c + 0.064083, y_c + -0.105376, z_c, rx, ry, rz], a, v)
    movel(p[x_c + 0.064017, y_c + -0.105334, z_c, rx, ry, rz], a, v)
    movel(p[x_c + 0.063951, y_c + -0.105292, z_c, rx, ry, rz], a, v)
    movel(p[x_c + 0.063887, y_c + -0.105251, z_c, rx, ry, rz], a, v)
    movel(p[x_c + 0.063823, y_c + -0.105211, z_c, rx, ry, rz], a, v)
    movel(p[x_c + 0.063761, y_c + -0.105171, z_c, rx, ry, rz], a, v)
    movel(p[x_c + 0.063699, y_c + -0.105131, z_c, rx, ry, rz], a, v)
    movel(p[x_c + 0.063639, y_c + -0.105093, z_c, rx, ry, rz], a, v)
    movel(p[x_c + 0.063580, y_c + -0.105055, z_c, rx, ry, rz], a, v)
    movel(p[x_c + 0.063522, y_c + -0.105018, z_c, rx, ry, rz], a, v)
    movel(p[x_c + 0.063465, y_c + -0.104981, z_c, rx, ry, rz], a, v)
    movel(p[x_c + 0.063410, y_c + -0.104946, z_c, rx, ry, rz], a, v)
    movel(p[x_c + 0.063410, y_c + -0.104946, z_c, rx, ry, rz], a, v)
    movel(p[x_c + 0.063355, y_c + -0.104911, z_c, rx, ry, rz], a, v)
    movel(p[x_c + 0.063301, y_c + -0.104876, z_c, rx, ry, rz], a, v)
    movel(p[x_c + 0.063247, y_c + -0.104842, z_c, rx, ry, rz], a, v)
    movel(p[x_c + 0.063194, y_c + -0.104808, z_c, rx, ry, rz], a, v)
    movel(p[x_c + 0.063141, y_c + -0.104775, z_c, rx, ry, rz], a, v)
    movel(p[x_c + 0.063089, y_c + -0.104742, z_c, rx, ry, rz], a, v)
    movel(p[x_c + 0.063037, y_c + -0.104709, z_c, rx, ry, rz], a, v)
    movel(p[x_c + 0.062986, y_c + -0.104677, z_c, rx, ry, rz], a, v)
    movel(p[x_c + 0.062935, y_c + -0.104645, z_c, rx, ry, rz], a, v)
    movel(p[x_c + 0.062885, y_c + -0.104614, z_c, rx, ry, rz], a, v)
    movel(p[x_c + 0.062835, y_c + -0.104584, z_c, rx, ry, rz], a, v)
    movel(p[x_c + 0.062786, y_c + -0.104554, z_c, rx, ry, rz], a, v)
    movel(p[x_c + 0.062738, y_c + -0.104524, z_c, rx, ry, rz], a, v)
    movel(p[x_c + 0.062691, y_c + -0.104495, z_c, rx, ry, rz], a, v)
    movel(p[x_c + 0.062644, y_c + -0.104467, z_c, rx, ry, rz], a, v)
    movel(p[x_c + 0.062598, y_c + -0.104439, z_c, rx, ry, rz], a, v)
    movel(p[x_c + 0.062553, y_c + -0.104412, z_c, rx, ry, rz], a, v)
    movel(p[x_c + 0.062509, y_c + -0.104385, z_c, rx, ry, rz], a, v)
    movel(p[x_c + 0.062465, y_c + -0.104359, z_c, rx, ry, rz], a, v)
    movel(p[x_c + 0.062423, y_c + -0.104334, z_c, rx, ry, rz], a, v)
    movel(p[x_c + 0.062381, y_c + -0.104309, z_c, rx, ry, rz], a, v)
    movel(p[x_c + 0.062341, y_c + -0.104285, z_c, rx, ry, rz], a, v)
    movel(p[x_c + 0.062301, y_c + -0.104262, z_c, rx, ry, rz], a, v)
    movel(p[x_c + 0.062262, y_c + -0.104240, z_c, rx, ry, rz], a, v)
    movel(p[x_c + 0.062225, y_c + -0.104218, z_c, rx, ry, rz], a, v)
    movel(p[x_c + 0.062189, y_c + -0.104197, z_c, rx, ry, rz], a, v)
    movel(p[x_c + 0.062153, y_c + -0.104177, z_c, rx, ry, rz], a, v)
    movel(p[x_c + 0.062119, y_c + -0.104158, z_c, rx, ry, rz], a, v)
    movel(p[x_c + 0.062086, y_c + -0.104139, z_c, rx, ry, rz], a, v)
    movel(p[x_c + 0.062054, y_c + -0.104122, z_c, rx, ry, rz], a, v)
    movel(p[x_c + 0.062024, y_c + -0.104105, z_c, rx, ry, rz], a, v)
    movel(p[x_c + 0.061994, y_c + -0.104089, z_c, rx, ry, rz], a, v)
    movel(p[x_c + 0.061966, y_c + -0.104074, z_c, rx, ry, rz], a, v)
    movel(p[x_c + 0.061940, y_c + -0.104060, z_c, rx, ry, rz], a, v)
    movel(p[x_c + 0.061914, y_c + -0.104047, z_c, rx, ry, rz], a, v)
    movel(p[x_c + 0.061891, y_c + -0.104034, z_c, rx, ry, rz], a, v)
    movel(p[x_c + 0.061868, y_c + -0.104023, z_c, rx, ry, rz], a, v)
    movel(p[x_c + 0.061847, y_c + -0.104013, z_c, rx, ry, rz], a, v)
    movel(p[x_c + 0.061827, y_c + -0.104003, z_c, rx, ry, rz], a, v)
    movel(p[x_c + 0.061809, y_c + -0.103995, z_c, rx, ry, rz], a, v)
    movel(p[x_c + 0.061793, y_c + -0.103988, z_c, rx, ry, rz], a, v)
    movel(p[x_c + 0.061778, y_c + -0.103982, z_c, rx, ry, rz], a, v)
    movel(p[x_c + 0.061764, y_c + -0.103977, z_c, rx, ry, rz], a, v)
    movel(p[x_c + 0.061753, y_c + -0.103973, z_c, rx, ry, rz], a, v)
    movel(p[x_c + 0.061743, y_c + -0.103970, z_c, rx, ry, rz], a, v)
    movel(p[x_c + 0.061734, y_c + -0.103968, z_c, rx, ry, rz], a, v)
    movel(p[x_c + 0.061728, y_c + -0.103967, z_c, rx, ry, rz], a, v)
    movel(p[x_c + 0.061723, y_c + -0.103968, z_c, rx, ry, rz], a, v)
    movel(p[x_c + 0.061720, y_c + -0.103969, z_c, rx, ry, rz], a, v)
    movel(p[x_c + 0.061720, y_c + -0.103969, z_c, rx, ry, rz], a, v)
    movel(p[x_c + 0.061718, y_c + -0.103976, z_c, rx, ry, rz], a, v)
    movel(p[x_c + 0.061721, y_c + -0.103988, z_c, rx, ry, rz], a, v)
    movel(p[x_c + 0.061730, y_c + -0.104005, z_c, rx, ry, rz], a, v)
    movel(p[x_c + 0.061744, y_c + -0.104026, z_c, rx, ry, rz], a, v)
    movel(p[x_c + 0.061763, y_c + -0.104051, z_c, rx, ry, rz], a, v)
    movel(p[x_c + 0.061787, y_c + -0.104081, z_c, rx, ry, rz], a, v)
    movel(p[x_c + 0.061815, y_c + -0.104116, z_c, rx, ry, rz], a, v)
    movel(p[x_c + 0.061849, y_c + -0.104154, z_c, rx, ry, rz], a, v)
    movel(p[x_c + 0.061887, y_c + -0.104196, z_c, rx, ry, rz], a, v)
    movel(p[x_c + 0.061929, y_c + -0.104242, z_c, rx, ry, rz], a, v)
    movel(p[x_c + 0.061976, y_c + -0.104292, z_c, rx, ry, rz], a, v)
    movel(p[x_c + 0.062026, y_c + -0.104346, z_c, rx, ry, rz], a, v)
    movel(p[x_c + 0.062081, y_c + -0.104403, z_c, rx, ry, rz], a, v)
    movel(p[x_c + 0.062140, y_c + -0.104464, z_c, rx, ry, rz], a, v)
    movel(p[x_c + 0.062203, y_c + -0.104528, z_c, rx, ry, rz], a, v)
    movel(p[x_c + 0.062270, y_c + -0.104595, z_c, rx, ry, rz], a, v)
    movel(p[x_c + 0.062340, y_c + -0.104666, z_c, rx, ry, rz], a, v)
    movel(p[x_c + 0.062414, y_c + -0.104739, z_c, rx, ry, rz], a, v)
    movel(p[x_c + 0.062491, y_c + -0.104815, z_c, rx, ry, rz], a, v)
    movel(p[x_c + 0.062571, y_c + -0.104895, z_c, rx, ry, rz], a, v)
    movel(p[x_c + 0.062654, y_c + -0.104976, z_c, rx, ry, rz], a, v)
    movel(p[x_c + 0.062741, y_c + -0.105061, z_c, rx, ry, rz], a, v)
    movel(p[x_c + 0.062830, y_c + -0.105147, z_c, rx, ry, rz], a, v)
    movel(p[x_c + 0.062923, y_c + -0.105236, z_c, rx, ry, rz], a, v)
    movel(p[x_c + 0.063018, y_c + -0.105328, z_c, rx, ry, rz], a, v)
    movel(p[x_c + 0.063115, y_c + -0.105421, z_c, rx, ry, rz], a, v)
    movel(p[x_c + 0.063215, y_c + -0.105517, z_c, rx, ry, rz], a, v)
    movel(p[x_c + 0.063318, y_c + -0.105614, z_c, rx, ry, rz], a, v)
    movel(p[x_c + 0.063422, y_c + -0.105713, z_c, rx, ry, rz], a, v)
    movel(p[x_c + 0.063529, y_c + -0.105814, z_c, rx, ry, rz], a, v)
    movel(p[x_c + 0.063638, y_c + -0.105916, z_c, rx, ry, rz], a, v)
    movel(p[x_c + 0.063748, y_c + -0.106020, z_c, rx, ry, rz], a, v)
    movel(p[x_c + 0.063860, y_c + -0.106125, z_c, rx, ry, rz], a, v)
    movel(p[x_c + 0.063974, y_c + -0.106231, z_c, rx, ry, rz], a, v)
    movel(p[x_c + 0.064090, y_c + -0.106338, z_c, rx, ry, rz], a, v)
    movel(p[x_c + 0.064207, y_c + -0.106447, z_c, rx, ry, rz], a, v)
    movel(p[x_c + 0.064325, y_c + -0.106556, z_c, rx, ry, rz], a, v)
    movel(p[x_c + 0.064444, y_c + -0.106666, z_c, rx, ry, rz], a, v)
    movel(p[x_c + 0.064565, y_c + -0.106776, z_c, rx, ry, rz], a, v)
    movel(p[x_c + 0.064686, y_c + -0.106888, z_c, rx, ry, rz], a, v)
    movel(p[x_c + 0.064808, y_c + -0.106999, z_c, rx, ry, rz], a, v)
    movel(p[x_c + 0.064931, y_c + -0.107111, z_c, rx, ry, rz], a, v)
    movel(p[x_c + 0.065055, y_c + -0.107223, z_c, rx, ry, rz], a, v)
    movel(p[x_c + 0.065179, y_c + -0.107335, z_c, rx, ry, rz], a, v)
    movel(p[x_c + 0.065303, y_c + -0.107448, z_c, rx, ry, rz], a, v)
    movel(p[x_c + 0.065428, y_c + -0.107560, z_c, rx, ry, rz], a, v)
    movel(p[x_c + 0.065552, y_c + -0.107671, z_c, rx, ry, rz], a, v)
    movel(p[x_c + 0.065677, y_c + -0.107783, z_c, rx, ry, rz], a, v)
    movel(p[x_c + 0.065802, y_c + -0.107894, z_c, rx, ry, rz], a, v)
    movel(p[x_c + 0.065802, y_c + -0.107894, z_c, rx, ry, rz], a, v)
    movel(p[x_c + 0.065880, y_c + -0.107964, z_c, rx, ry, rz], a, v)
    movel(p[x_c + 0.065956, y_c + -0.108031, z_c, rx, ry, rz], a, v)
    movel(p[x_c + 0.066029, y_c + -0.108097, z_c, rx, ry, rz], a, v)
    movel(p[x_c + 0.066101, y_c + -0.108162, z_c, rx, ry, rz], a, v)
    movel(p[x_c + 0.066169, y_c + -0.108224, z_c, rx, ry, rz], a, v)
    movel(p[x_c + 0.066236, y_c + -0.108284, z_c, rx, ry, rz], a, v)
    movel(p[x_c + 0.066300, y_c + -0.108343, z_c, rx, ry, rz], a, v)
    movel(p[x_c + 0.066362, y_c + -0.108400, z_c, rx, ry, rz], a, v)
    movel(p[x_c + 0.066422, y_c + -0.108456, z_c, rx, ry, rz], a, v)
    movel(p[x_c + 0.066480, y_c + -0.108509, z_c, rx, ry, rz], a, v)
    movel(p[x_c + 0.066535, y_c + -0.108561, z_c, rx, ry, rz], a, v)
    movel(p[x_c + 0.066588, y_c + -0.108611, z_c, rx, ry, rz], a, v)
    movel(p[x_c + 0.066639, y_c + -0.108660, z_c, rx, ry, rz], a, v)
    movel(p[x_c + 0.066688, y_c + -0.108707, z_c, rx, ry, rz], a, v)
    movel(p[x_c + 0.066735, y_c + -0.108752, z_c, rx, ry, rz], a, v)
    movel(p[x_c + 0.066779, y_c + -0.108796, z_c, rx, ry, rz], a, v)
    movel(p[x_c + 0.066821, y_c + -0.108838, z_c, rx, ry, rz], a, v)
    movel(p[x_c + 0.066862, y_c + -0.108878, z_c, rx, ry, rz], a, v)
    movel(p[x_c + 0.066900, y_c + -0.108917, z_c, rx, ry, rz], a, v)
    movel(p[x_c + 0.066936, y_c + -0.108954, z_c, rx, ry, rz], a, v)
    movel(p[x_c + 0.066970, y_c + -0.108990, z_c, rx, ry, rz], a, v)
    movel(p[x_c + 0.067002, y_c + -0.109025, z_c, rx, ry, rz], a, v)
    movel(p[x_c + 0.067032, y_c + -0.109058, z_c, rx, ry, rz], a, v)
    movel(p[x_c + 0.067060, y_c + -0.109089, z_c, rx, ry, rz], a, v)
    movel(p[x_c + 0.067086, y_c + -0.109119, z_c, rx, ry, rz], a, v)
    movel(p[x_c + 0.067109, y_c + -0.109147, z_c, rx, ry, rz], a, v)
    movel(p[x_c + 0.067131, y_c + -0.109175, z_c, rx, ry, rz], a, v)
    movel(p[x_c + 0.067151, y_c + -0.109200, z_c, rx, ry, rz], a, v)
    movel(p[x_c + 0.067169, y_c + -0.109225, z_c, rx, ry, rz], a, v)
    movel(p[x_c + 0.067185, y_c + -0.109248, z_c, rx, ry, rz], a, v)
    movel(p[x_c + 0.067200, y_c + -0.109269, z_c, rx, ry, rz], a, v)
    movel(p[x_c + 0.067212, y_c + -0.109290, z_c, rx, ry, rz], a, v)
    movel(p[x_c + 0.067222, y_c + -0.109309, z_c, rx, ry, rz], a, v)
    movel(p[x_c + 0.067231, y_c + -0.109326, z_c, rx, ry, rz], a, v)
    movel(p[x_c + 0.067238, y_c + -0.109343, z_c, rx, ry, rz], a, v)
    movel(p[x_c + 0.067242, y_c + -0.109358, z_c, rx, ry, rz], a, v)
    movel(p[x_c + 0.067245, y_c + -0.109372, z_c, rx, ry, rz], a, v)
    movel(p[x_c + 0.067247, y_c + -0.109385, z_c, rx, ry, rz], a, v)
    movel(p[x_c + 0.067246, y_c + -0.109396, z_c, rx, ry, rz], a, v)
    movel(p[x_c + 0.067244, y_c + -0.109406, z_c, rx, ry, rz], a, v)
    movel(p[x_c + 0.067240, y_c + -0.109416, z_c, rx, ry, rz], a, v)
    movel(p[x_c + 0.067234, y_c + -0.109424, z_c, rx, ry, rz], a, v)
    movel(p[x_c + 0.067226, y_c + -0.109431, z_c, rx, ry, rz], a, v)
    movel(p[x_c + 0.067217, y_c + -0.109436, z_c, rx, ry, rz], a, v)
    movel(p[x_c + 0.067206, y_c + -0.109441, z_c, rx, ry, rz], a, v)
    movel(p[x_c + 0.067194, y_c + -0.109445, z_c, rx, ry, rz], a, v)
    movel(p[x_c + 0.067179, y_c + -0.109447, z_c, rx, ry, rz], a, v)
    movel(p[x_c + 0.067163, y_c + -0.109449, z_c, rx, ry, rz], a, v)
    movel(p[x_c + 0.067146, y_c + -0.109449, z_c, rx, ry, rz], a, v)
    movel(p[x_c + 0.067146, y_c + -0.109449, z_c, rx, ry, rz], a, v)
    movel(p[x_c + 0.067139, y_c + -0.109448, z_c, rx, ry, rz], a, v)
    movel(p[x_c + 0.067129, y_c + -0.109445, z_c, rx, ry, rz], a, v)
    movel(p[x_c + 0.067117, y_c + -0.109440, z_c, rx, ry, rz], a, v)
    movel(p[x_c + 0.067101, y_c + -0.109432, z_c, rx, ry, rz], a, v)
    movel(p[x_c + 0.067082, y_c + -0.109423, z_c, rx, ry, rz], a, v)
    movel(p[x_c + 0.067059, y_c + -0.109411, z_c, rx, ry, rz], a, v)
    movel(p[x_c + 0.067034, y_c + -0.109398, z_c, rx, ry, rz], a, v)
    movel(p[x_c + 0.067007, y_c + -0.109383, z_c, rx, ry, rz], a, v)
    movel(p[x_c + 0.066976, y_c + -0.109366, z_c, rx, ry, rz], a, v)
    movel(p[x_c + 0.066942, y_c + -0.109346, z_c, rx, ry, rz], a, v)
    movel(p[x_c + 0.066906, y_c + -0.109326, z_c, rx, ry, rz], a, v)
    movel(p[x_c + 0.066867, y_c + -0.109303, z_c, rx, ry, rz], a, v)
    movel(p[x_c + 0.066826, y_c + -0.109279, z_c, rx, ry, rz], a, v)
    movel(p[x_c + 0.066782, y_c + -0.109252, z_c, rx, ry, rz], a, v)
    movel(p[x_c + 0.066735, y_c + -0.109225, z_c, rx, ry, rz], a, v)
    movel(p[x_c + 0.066686, y_c + -0.109195, z_c, rx, ry, rz], a, v)
    movel(p[x_c + 0.066635, y_c + -0.109164, z_c, rx, ry, rz], a, v)
    movel(p[x_c + 0.066581, y_c + -0.109131, z_c, rx, ry, rz], a, v)
    movel(p[x_c + 0.066525, y_c + -0.109097, z_c, rx, ry, rz], a, v)
    movel(p[x_c + 0.066467, y_c + -0.109061, z_c, rx, ry, rz], a, v)
    movel(p[x_c + 0.066406, y_c + -0.109024, z_c, rx, ry, rz], a, v)
    movel(p[x_c + 0.066344, y_c + -0.108985, z_c, rx, ry, rz], a, v)
    movel(p[x_c + 0.066279, y_c + -0.108945, z_c, rx, ry, rz], a, v)
    movel(p[x_c + 0.066213, y_c + -0.108904, z_c, rx, ry, rz], a, v)
    movel(p[x_c + 0.066144, y_c + -0.108861, z_c, rx, ry, rz], a, v)
    movel(p[x_c + 0.066074, y_c + -0.108817, z_c, rx, ry, rz], a, v)
    movel(p[x_c + 0.066002, y_c + -0.108771, z_c, rx, ry, rz], a, v)
    movel(p[x_c + 0.065928, y_c + -0.108725, z_c, rx, ry, rz], a, v)
    movel(p[x_c + 0.065852, y_c + -0.108677, z_c, rx, ry, rz], a, v)
    movel(p[x_c + 0.065774, y_c + -0.108628, z_c, rx, ry, rz], a, v)
    movel(p[x_c + 0.065695, y_c + -0.108578, z_c, rx, ry, rz], a, v)
    movel(p[x_c + 0.065615, y_c + -0.108526, z_c, rx, ry, rz], a, v)
    movel(p[x_c + 0.065532, y_c + -0.108474, z_c, rx, ry, rz], a, v)
    movel(p[x_c + 0.065449, y_c + -0.108421, z_c, rx, ry, rz], a, v)
    movel(p[x_c + 0.065364, y_c + -0.108366, z_c, rx, ry, rz], a, v)
    movel(p[x_c + 0.065277, y_c + -0.108311, z_c, rx, ry, rz], a, v)
    movel(p[x_c + 0.065190, y_c + -0.108255, z_c, rx, ry, rz], a, v)
    movel(p[x_c + 0.065101, y_c + -0.108198, z_c, rx, ry, rz], a, v)
    movel(p[x_c + 0.065011, y_c + -0.108140, z_c, rx, ry, rz], a, v)
    movel(p[x_c + 0.064920, y_c + -0.108081, z_c, rx, ry, rz], a, v)
    movel(p[x_c + 0.064827, y_c + -0.108021, z_c, rx, ry, rz], a, v)
    movel(p[x_c + 0.064734, y_c + -0.107961, z_c, rx, ry, rz], a, v)
    movel(p[x_c + 0.064640, y_c + -0.107900, z_c, rx, ry, rz], a, v)
    movel(p[x_c + 0.064545, y_c + -0.107838, z_c, rx, ry, rz], a, v)
    movel(p[x_c + 0.064449, y_c + -0.107776, z_c, rx, ry, rz], a, v)
    movel(p[x_c + 0.064352, y_c + -0.107712, z_c, rx, ry, rz], a, v)
    movel(p[x_c + 0.064255, y_c + -0.107649, z_c, rx, ry, rz], a, v)
    movel(p[x_c + 0.064156, y_c + -0.107585, z_c, rx, ry, rz], a, v)
    movel(p[x_c + 0.064058, y_c + -0.107520, z_c, rx, ry, rz], a, v)
    movel(p[x_c + 0.064058, y_c + -0.107520, z_c, rx, ry, rz], a, v)
    movel(p[x_c + 0.063844, y_c + -0.107380, z_c, rx, ry, rz], a, v)
    movel(p[x_c + 0.063630, y_c + -0.107241, z_c, rx, ry, rz], a, v)
    movel(p[x_c + 0.063415, y_c + -0.107101, z_c, rx, ry, rz], a, v)
    movel(p[x_c + 0.063200, y_c + -0.106962, z_c, rx, ry, rz], a, v)
    movel(p[x_c + 0.062985, y_c + -0.106823, z_c, rx, ry, rz], a, v)
    movel(p[x_c + 0.062769, y_c + -0.106685, z_c, rx, ry, rz], a, v)
    movel(p[x_c + 0.062555, y_c + -0.106547, z_c, rx, ry, rz], a, v)
    movel(p[x_c + 0.062340, y_c + -0.106410, z_c, rx, ry, rz], a, v)
    movel(p[x_c + 0.062127, y_c + -0.106274, z_c, rx, ry, rz], a, v)
    movel(p[x_c + 0.061914, y_c + -0.106140, z_c, rx, ry, rz], a, v)
    movel(p[x_c + 0.061703, y_c + -0.106006, z_c, rx, ry, rz], a, v)
    movel(p[x_c + 0.061494, y_c + -0.105874, z_c, rx, ry, rz], a, v)
    movel(p[x_c + 0.061286, y_c + -0.105743, z_c, rx, ry, rz], a, v)
    movel(p[x_c + 0.061080, y_c + -0.105614, z_c, rx, ry, rz], a, v)
    movel(p[x_c + 0.060876, y_c + -0.105487, z_c, rx, ry, rz], a, v)
    movel(p[x_c + 0.060674, y_c + -0.105362, z_c, rx, ry, rz], a, v)
    movel(p[x_c + 0.060476, y_c + -0.105238, z_c, rx, ry, rz], a, v)
    movel(p[x_c + 0.060280, y_c + -0.105117, z_c, rx, ry, rz], a, v)
    movel(p[x_c + 0.060087, y_c + -0.104999, z_c, rx, ry, rz], a, v)
    movel(p[x_c + 0.059897, y_c + -0.104882, z_c, rx, ry, rz], a, v)
    movel(p[x_c + 0.059711, y_c + -0.104769, z_c, rx, ry, rz], a, v)
    movel(p[x_c + 0.059529, y_c + -0.104658, z_c, rx, ry, rz], a, v)
    movel(p[x_c + 0.059351, y_c + -0.104550, z_c, rx, ry, rz], a, v)
    movel(p[x_c + 0.059177, y_c + -0.104445, z_c, rx, ry, rz], a, v)
    movel(p[x_c + 0.059008, y_c + -0.104343, z_c, rx, ry, rz], a, v)
    movel(p[x_c + 0.058843, y_c + -0.104244, z_c, rx, ry, rz], a, v)
    movel(p[x_c + 0.058683, y_c + -0.104149, z_c, rx, ry, rz], a, v)
    movel(p[x_c + 0.058528, y_c + -0.104058, z_c, rx, ry, rz], a, v)
    movel(p[x_c + 0.058379, y_c + -0.103970, z_c, rx, ry, rz], a, v)
    movel(p[x_c + 0.058235, y_c + -0.103886, z_c, rx, ry, rz], a, v)
    movel(p[x_c + 0.058097, y_c + -0.103806, z_c, rx, ry, rz], a, v)
    movel(p[x_c + 0.057966, y_c + -0.103730, z_c, rx, ry, rz], a, v)
    movel(p[x_c + 0.057840, y_c + -0.103658, z_c, rx, ry, rz], a, v)
    movel(p[x_c + 0.057721, y_c + -0.103591, z_c, rx, ry, rz], a, v)
    movel(p[x_c + 0.057609, y_c + -0.103528, z_c, rx, ry, rz], a, v)
    movel(p[x_c + 0.057504, y_c + -0.103470, z_c, rx, ry, rz], a, v)
    movel(p[x_c + 0.057406, y_c + -0.103417, z_c, rx, ry, rz], a, v)
    movel(p[x_c + 0.057315, y_c + -0.103368, z_c, rx, ry, rz], a, v)
    movel(p[x_c + 0.057232, y_c + -0.103325, z_c, rx, ry, rz], a, v)
    movel(p[x_c + 0.057157, y_c + -0.103287, z_c, rx, ry, rz], a, v)
    movel(p[x_c + 0.057090, y_c + -0.103254, z_c, rx, ry, rz], a, v)
    movel(p[x_c + 0.057032, y_c + -0.103227, z_c, rx, ry, rz], a, v)
    movel(p[x_c + 0.056982, y_c + -0.103206, z_c, rx, ry, rz], a, v)
    movel(p[x_c + 0.056940, y_c + -0.103190, z_c, rx, ry, rz], a, v)
    movel(p[x_c + 0.056908, y_c + -0.103180, z_c, rx, ry, rz], a, v)
    movel(p[x_c + 0.056886, y_c + -0.103176, z_c, rx, ry, rz], a, v)
    movel(p[x_c + 0.056872, y_c + -0.103179, z_c, rx, ry, rz], a, v)
    movel(p[x_c + 0.056869, y_c + -0.103187, z_c, rx, ry, rz], a, v)
    movel(p[x_c + 0.056875, y_c + -0.103202, z_c, rx, ry, rz], a, v)
    movel(p[x_c + 0.056875, y_c + -0.103202, z_c, rx, ry, rz], a, v)
    movel(p[x_c + 0.056880, y_c + -0.103210, z_c, rx, ry, rz], a, v)
    movel(p[x_c + 0.056887, y_c + -0.103219, z_c, rx, ry, rz], a, v)
    movel(p[x_c + 0.056895, y_c + -0.103229, z_c, rx, ry, rz], a, v)
    movel(p[x_c + 0.056905, y_c + -0.103240, z_c, rx, ry, rz], a, v)
    movel(p[x_c + 0.056916, y_c + -0.103252, z_c, rx, ry, rz], a, v)
    movel(p[x_c + 0.056929, y_c + -0.103265, z_c, rx, ry, rz], a, v)
    movel(p[x_c + 0.056943, y_c + -0.103278, z_c, rx, ry, rz], a, v)
    movel(p[x_c + 0.056959, y_c + -0.103293, z_c, rx, ry, rz], a, v)
    movel(p[x_c + 0.056976, y_c + -0.103309, z_c, rx, ry, rz], a, v)
    movel(p[x_c + 0.056994, y_c + -0.103326, z_c, rx, ry, rz], a, v)
    movel(p[x_c + 0.057014, y_c + -0.103343, z_c, rx, ry, rz], a, v)
    movel(p[x_c + 0.057035, y_c + -0.103362, z_c, rx, ry, rz], a, v)
    movel(p[x_c + 0.057057, y_c + -0.103381, z_c, rx, ry, rz], a, v)
    movel(p[x_c + 0.057080, y_c + -0.103401, z_c, rx, ry, rz], a, v)
    movel(p[x_c + 0.057105, y_c + -0.103422, z_c, rx, ry, rz], a, v)
    movel(p[x_c + 0.057131, y_c + -0.103444, z_c, rx, ry, rz], a, v)
    movel(p[x_c + 0.057158, y_c + -0.103466, z_c, rx, ry, rz], a, v)
    movel(p[x_c + 0.057186, y_c + -0.103490, z_c, rx, ry, rz], a, v)
    movel(p[x_c + 0.057215, y_c + -0.103513, z_c, rx, ry, rz], a, v)
    movel(p[x_c + 0.057245, y_c + -0.103538, z_c, rx, ry, rz], a, v)
    movel(p[x_c + 0.057277, y_c + -0.103563, z_c, rx, ry, rz], a, v)
    movel(p[x_c + 0.057309, y_c + -0.103589, z_c, rx, ry, rz], a, v)
    movel(p[x_c + 0.057342, y_c + -0.103616, z_c, rx, ry, rz], a, v)
    movel(p[x_c + 0.057376, y_c + -0.103643, z_c, rx, ry, rz], a, v)
    movel(p[x_c + 0.057411, y_c + -0.103671, z_c, rx, ry, rz], a, v)
    movel(p[x_c + 0.057447, y_c + -0.103699, z_c, rx, ry, rz], a, v)
    movel(p[x_c + 0.057484, y_c + -0.103728, z_c, rx, ry, rz], a, v)
    movel(p[x_c + 0.057522, y_c + -0.103757, z_c, rx, ry, rz], a, v)
    movel(p[x_c + 0.057560, y_c + -0.103787, z_c, rx, ry, rz], a, v)
    movel(p[x_c + 0.057600, y_c + -0.103817, z_c, rx, ry, rz], a, v)
    movel(p[x_c + 0.057640, y_c + -0.103848, z_c, rx, ry, rz], a, v)
    movel(p[x_c + 0.057680, y_c + -0.103879, z_c, rx, ry, rz], a, v)
    movel(p[x_c + 0.057722, y_c + -0.103910, z_c, rx, ry, rz], a, v)
    movel(p[x_c + 0.057764, y_c + -0.103942, z_c, rx, ry, rz], a, v)
    movel(p[x_c + 0.057807, y_c + -0.103974, z_c, rx, ry, rz], a, v)
    movel(p[x_c + 0.057850, y_c + -0.104007, z_c, rx, ry, rz], a, v)
    movel(p[x_c + 0.057894, y_c + -0.104040, z_c, rx, ry, rz], a, v)
    movel(p[x_c + 0.057938, y_c + -0.104073, z_c, rx, ry, rz], a, v)
    movel(p[x_c + 0.057983, y_c + -0.104106, z_c, rx, ry, rz], a, v)
    movel(p[x_c + 0.058029, y_c + -0.104140, z_c, rx, ry, rz], a, v)
    movel(p[x_c + 0.058075, y_c + -0.104174, z_c, rx, ry, rz], a, v)
    movel(p[x_c + 0.058121, y_c + -0.104208, z_c, rx, ry, rz], a, v)
    movel(p[x_c + 0.058168, y_c + -0.104242, z_c, rx, ry, rz], a, v)
    movel(p[x_c + 0.058215, y_c + -0.104277, z_c, rx, ry, rz], a, v)
    movel(p[x_c + 0.058263, y_c + -0.104311, z_c, rx, ry, rz], a, v)
    movel(p[x_c + 0.058311, y_c + -0.104346, z_c, rx, ry, rz], a, v)
    movel(p[x_c + 0.058359, y_c + -0.104381, z_c, rx, ry, rz], a, v)
    movel(p[x_c + 0.058408, y_c + -0.104415, z_c, rx, ry, rz], a, v)
    movel(p[x_c + 0.058456, y_c + -0.104450, z_c, rx, ry, rz], a, v)
    movel(p[x_c + 0.058456, y_c + -0.104450, z_c, rx, ry, rz], a, v)
    movel(p[x_c + 0.058505, y_c + -0.104485, z_c, rx, ry, rz], a, v)
    movel(p[x_c + 0.058553, y_c + -0.104520, z_c, rx, ry, rz], a, v)
    movel(p[x_c + 0.058600, y_c + -0.104554, z_c, rx, ry, rz], a, v)
    movel(p[x_c + 0.058647, y_c + -0.104588, z_c, rx, ry, rz], a, v)
    movel(p[x_c + 0.058694, y_c + -0.104622, z_c, rx, ry, rz], a, v)
    movel(p[x_c + 0.058740, y_c + -0.104656, z_c, rx, ry, rz], a, v)
    movel(p[x_c + 0.058785, y_c + -0.104690, z_c, rx, ry, rz], a, v)
    movel(p[x_c + 0.058829, y_c + -0.104723, z_c, rx, ry, rz], a, v)
    movel(p[x_c + 0.058873, y_c + -0.104756, z_c, rx, ry, rz], a, v)
    movel(p[x_c + 0.058916, y_c + -0.104789, z_c, rx, ry, rz], a, v)
    movel(p[x_c + 0.058959, y_c + -0.104821, z_c, rx, ry, rz], a, v)
    movel(p[x_c + 0.059000, y_c + -0.104853, z_c, rx, ry, rz], a, v)
    movel(p[x_c + 0.059041, y_c + -0.104884, z_c, rx, ry, rz], a, v)
    movel(p[x_c + 0.059081, y_c + -0.104916, z_c, rx, ry, rz], a, v)
    movel(p[x_c + 0.059121, y_c + -0.104946, z_c, rx, ry, rz], a, v)
    movel(p[x_c + 0.059159, y_c + -0.104977, z_c, rx, ry, rz], a, v)
    movel(p[x_c + 0.059196, y_c + -0.105007, z_c, rx, ry, rz], a, v)
    movel(p[x_c + 0.059233, y_c + -0.105036, z_c, rx, ry, rz], a, v)
    movel(p[x_c + 0.059269, y_c + -0.105065, z_c, rx, ry, rz], a, v)
    movel(p[x_c + 0.059304, y_c + -0.105093, z_c, rx, ry, rz], a, v)
    movel(p[x_c + 0.059337, y_c + -0.105121, z_c, rx, ry, rz], a, v)
    movel(p[x_c + 0.059370, y_c + -0.105148, z_c, rx, ry, rz], a, v)
    movel(p[x_c + 0.059402, y_c + -0.105175, z_c, rx, ry, rz], a, v)
    movel(p[x_c + 0.059433, y_c + -0.105201, z_c, rx, ry, rz], a, v)
    movel(p[x_c + 0.059462, y_c + -0.105226, z_c, rx, ry, rz], a, v)
    movel(p[x_c + 0.059491, y_c + -0.105251, z_c, rx, ry, rz], a, v)
    movel(p[x_c + 0.059518, y_c + -0.105275, z_c, rx, ry, rz], a, v)
    movel(p[x_c + 0.059545, y_c + -0.105299, z_c, rx, ry, rz], a, v)
    movel(p[x_c + 0.059570, y_c + -0.105322, z_c, rx, ry, rz], a, v)
    movel(p[x_c + 0.059594, y_c + -0.105344, z_c, rx, ry, rz], a, v)
    movel(p[x_c + 0.059617, y_c + -0.105365, z_c, rx, ry, rz], a, v)
    movel(p[x_c + 0.059639, y_c + -0.105385, z_c, rx, ry, rz], a, v)
    movel(p[x_c + 0.059659, y_c + -0.105405, z_c, rx, ry, rz], a, v)
    movel(p[x_c + 0.059678, y_c + -0.105424, z_c, rx, ry, rz], a, v)
    movel(p[x_c + 0.059696, y_c + -0.105442, z_c, rx, ry, rz], a, v)
    movel(p[x_c + 0.059712, y_c + -0.105459, z_c, rx, ry, rz], a, v)
    movel(p[x_c + 0.059727, y_c + -0.105476, z_c, rx, ry, rz], a, v)
    movel(p[x_c + 0.059741, y_c + -0.105491, z_c, rx, ry, rz], a, v)
    movel(p[x_c + 0.059753, y_c + -0.105506, z_c, rx, ry, rz], a, v)
    movel(p[x_c + 0.059764, y_c + -0.105519, z_c, rx, ry, rz], a, v)
    movel(p[x_c + 0.059774, y_c + -0.105532, z_c, rx, ry, rz], a, v)
    movel(p[x_c + 0.059782, y_c + -0.105544, z_c, rx, ry, rz], a, v)
    movel(p[x_c + 0.059788, y_c + -0.105555, z_c, rx, ry, rz], a, v)
    movel(p[x_c + 0.059793, y_c + -0.105564, z_c, rx, ry, rz], a, v)
    movel(p[x_c + 0.059797, y_c + -0.105573, z_c, rx, ry, rz], a, v)
    movel(p[x_c + 0.059799, y_c + -0.105581, z_c, rx, ry, rz], a, v)
    movel(p[x_c + 0.059799, y_c + -0.105587, z_c, rx, ry, rz], a, v)
    movel(p[x_c + 0.059798, y_c + -0.105592, z_c, rx, ry, rz], a, v)
    movel(p[x_c + 0.059795, y_c + -0.105597, z_c, rx, ry, rz], a, v)
    movel(p[x_c + 0.059795, y_c + -0.105597, z_c, rx, ry, rz], a, v)
    movel(p[x_c + 0.059786, y_c + -0.105602, z_c, rx, ry, rz], a, v)
    movel(p[x_c + 0.059774, y_c + -0.105605, z_c, rx, ry, rz], a, v)
    movel(p[x_c + 0.059759, y_c + -0.105605, z_c, rx, ry, rz], a, v)
    movel(p[x_c + 0.059740, y_c + -0.105603, z_c, rx, ry, rz], a, v)
    movel(p[x_c + 0.059717, y_c + -0.105599, z_c, rx, ry, rz], a, v)
    movel(p[x_c + 0.059691, y_c + -0.105593, z_c, rx, ry, rz], a, v)
    movel(p[x_c + 0.059662, y_c + -0.105584, z_c, rx, ry, rz], a, v)
    movel(p[x_c + 0.059630, y_c + -0.105574, z_c, rx, ry, rz], a, v)
    movel(p[x_c + 0.059595, y_c + -0.105562, z_c, rx, ry, rz], a, v)
    movel(p[x_c + 0.059557, y_c + -0.105548, z_c, rx, ry, rz], a, v)
    movel(p[x_c + 0.059516, y_c + -0.105532, z_c, rx, ry, rz], a, v)
    movel(p[x_c + 0.059473, y_c + -0.105514, z_c, rx, ry, rz], a, v)
    movel(p[x_c + 0.059428, y_c + -0.105495, z_c, rx, ry, rz], a, v)
    movel(p[x_c + 0.059380, y_c + -0.105474, z_c, rx, ry, rz], a, v)
    movel(p[x_c + 0.059330, y_c + -0.105452, z_c, rx, ry, rz], a, v)
    movel(p[x_c + 0.059278, y_c + -0.105428, z_c, rx, ry, rz], a, v)
    movel(p[x_c + 0.059223, y_c + -0.105402, z_c, rx, ry, rz], a, v)
    movel(p[x_c + 0.059167, y_c + -0.105375, z_c, rx, ry, rz], a, v)
    movel(p[x_c + 0.059110, y_c + -0.105347, z_c, rx, ry, rz], a, v)
    movel(p[x_c + 0.059051, y_c + -0.105318, z_c, rx, ry, rz], a, v)
    movel(p[x_c + 0.058990, y_c + -0.105288, z_c, rx, ry, rz], a, v)
    movel(p[x_c + 0.058928, y_c + -0.105256, z_c, rx, ry, rz], a, v)
    movel(p[x_c + 0.058865, y_c + -0.105224, z_c, rx, ry, rz], a, v)
    movel(p[x_c + 0.058800, y_c + -0.105190, z_c, rx, ry, rz], a, v)
    movel(p[x_c + 0.058735, y_c + -0.105156, z_c, rx, ry, rz], a, v)
    movel(p[x_c + 0.058669, y_c + -0.105121, z_c, rx, ry, rz], a, v)
    movel(p[x_c + 0.058602, y_c + -0.105085, z_c, rx, ry, rz], a, v)
    movel(p[x_c + 0.058534, y_c + -0.105048, z_c, rx, ry, rz], a, v)
    movel(p[x_c + 0.058466, y_c + -0.105011, z_c, rx, ry, rz], a, v)
    movel(p[x_c + 0.058398, y_c + -0.104973, z_c, rx, ry, rz], a, v)
    movel(p[x_c + 0.058330, y_c + -0.104934, z_c, rx, ry, rz], a, v)
    movel(p[x_c + 0.058261, y_c + -0.104895, z_c, rx, ry, rz], a, v)
    movel(p[x_c + 0.058192, y_c + -0.104856, z_c, rx, ry, rz], a, v)
    movel(p[x_c + 0.058124, y_c + -0.104817, z_c, rx, ry, rz], a, v)
    movel(p[x_c + 0.058055, y_c + -0.104777, z_c, rx, ry, rz], a, v)
    movel(p[x_c + 0.057988, y_c + -0.104737, z_c, rx, ry, rz], a, v)
    movel(p[x_c + 0.057920, y_c + -0.104696, z_c, rx, ry, rz], a, v)
    movel(p[x_c + 0.057853, y_c + -0.104656, z_c, rx, ry, rz], a, v)
    movel(p[x_c + 0.057787, y_c + -0.104616, z_c, rx, ry, rz], a, v)
    movel(p[x_c + 0.057722, y_c + -0.104576, z_c, rx, ry, rz], a, v)
    movel(p[x_c + 0.057658, y_c + -0.104536, z_c, rx, ry, rz], a, v)
    movel(p[x_c + 0.057595, y_c + -0.104496, z_c, rx, ry, rz], a, v)
    movel(p[x_c + 0.057533, y_c + -0.104456, z_c, rx, ry, rz], a, v)
    movel(p[x_c + 0.057473, y_c + -0.104417, z_c, rx, ry, rz], a, v)
    movel(p[x_c + 0.057414, y_c + -0.104378, z_c, rx, ry, rz], a, v)
    movel(p[x_c + 0.057356, y_c + -0.104340, z_c, rx, ry, rz], a, v)
    movel(p[x_c + 0.057301, y_c + -0.104302, z_c, rx, ry, rz], a, v)
    movel(p[x_c + 0.057247, y_c + -0.104265, z_c, rx, ry, rz], a, v)
    movel(p[x_c + 0.057195, y_c + -0.104228, z_c, rx, ry, rz], a, v)
    movel(p[x_c + 0.057195, y_c + -0.104228, z_c, rx, ry, rz], a, v)
    movel(p[x_c + 0.057184, y_c + -0.104220, z_c, rx, ry, rz], a, v)
    movel(p[x_c + 0.057173, y_c + -0.104213, z_c, rx, ry, rz], a, v)
    movel(p[x_c + 0.057164, y_c + -0.104206, z_c, rx, ry, rz], a, v)
    movel(p[x_c + 0.057155, y_c + -0.104201, z_c, rx, ry, rz], a, v)
    movel(p[x_c + 0.057147, y_c + -0.104196, z_c, rx, ry, rz], a, v)
    movel(p[x_c + 0.057140, y_c + -0.104192, z_c, rx, ry, rz], a, v)
    movel(p[x_c + 0.057134, y_c + -0.104188, z_c, rx, ry, rz], a, v)
    movel(p[x_c + 0.057128, y_c + -0.104185, z_c, rx, ry, rz], a, v)
    movel(p[x_c + 0.057124, y_c + -0.104183, z_c, rx, ry, rz], a, v)
    movel(p[x_c + 0.057120, y_c + -0.104182, z_c, rx, ry, rz], a, v)
    movel(p[x_c + 0.057117, y_c + -0.104181, z_c, rx, ry, rz], a, v)
    movel(p[x_c + 0.057115, y_c + -0.104181, z_c, rx, ry, rz], a, v)
    movel(p[x_c + 0.057113, y_c + -0.104182, z_c, rx, ry, rz], a, v)
    movel(p[x_c + 0.057113, y_c + -0.104183, z_c, rx, ry, rz], a, v)
    movel(p[x_c + 0.057113, y_c + -0.104185, z_c, rx, ry, rz], a, v)
    movel(p[x_c + 0.057114, y_c + -0.104188, z_c, rx, ry, rz], a, v)
    movel(p[x_c + 0.057115, y_c + -0.104191, z_c, rx, ry, rz], a, v)
    movel(p[x_c + 0.057118, y_c + -0.104195, z_c, rx, ry, rz], a, v)
    movel(p[x_c + 0.057121, y_c + -0.104199, z_c, rx, ry, rz], a, v)
    movel(p[x_c + 0.057125, y_c + -0.104205, z_c, rx, ry, rz], a, v)
    movel(p[x_c + 0.057129, y_c + -0.104210, z_c, rx, ry, rz], a, v)
    movel(p[x_c + 0.057135, y_c + -0.104217, z_c, rx, ry, rz], a, v)
    movel(p[x_c + 0.057141, y_c + -0.104224, z_c, rx, ry, rz], a, v)
    movel(p[x_c + 0.057147, y_c + -0.104232, z_c, rx, ry, rz], a, v)
    movel(p[x_c + 0.057155, y_c + -0.104240, z_c, rx, ry, rz], a, v)
    movel(p[x_c + 0.057163, y_c + -0.104249, z_c, rx, ry, rz], a, v)
    movel(p[x_c + 0.057172, y_c + -0.104258, z_c, rx, ry, rz], a, v)
    movel(p[x_c + 0.057181, y_c + -0.104268, z_c, rx, ry, rz], a, v)
    movel(p[x_c + 0.057192, y_c + -0.104279, z_c, rx, ry, rz], a, v)
    movel(p[x_c + 0.057203, y_c + -0.104290, z_c, rx, ry, rz], a, v)
    movel(p[x_c + 0.057214, y_c + -0.104302, z_c, rx, ry, rz], a, v)
    movel(p[x_c + 0.057226, y_c + -0.104314, z_c, rx, ry, rz], a, v)
    movel(p[x_c + 0.057239, y_c + -0.104327, z_c, rx, ry, rz], a, v)
    movel(p[x_c + 0.057253, y_c + -0.104341, z_c, rx, ry, rz], a, v)
    movel(p[x_c + 0.057267, y_c + -0.104355, z_c, rx, ry, rz], a, v)
    movel(p[x_c + 0.057282, y_c + -0.104369, z_c, rx, ry, rz], a, v)
    movel(p[x_c + 0.057297, y_c + -0.104384, z_c, rx, ry, rz], a, v)
    movel(p[x_c + 0.057313, y_c + -0.104400, z_c, rx, ry, rz], a, v)
    movel(p[x_c + 0.057330, y_c + -0.104416, z_c, rx, ry, rz], a, v)
    movel(p[x_c + 0.057347, y_c + -0.104432, z_c, rx, ry, rz], a, v)
    movel(p[x_c + 0.057365, y_c + -0.104449, z_c, rx, ry, rz], a, v)
    movel(p[x_c + 0.057384, y_c + -0.104467, z_c, rx, ry, rz], a, v)
    movel(p[x_c + 0.057403, y_c + -0.104485, z_c, rx, ry, rz], a, v)
    movel(p[x_c + 0.057423, y_c + -0.104503, z_c, rx, ry, rz], a, v)
    movel(p[x_c + 0.057443, y_c + -0.104522, z_c, rx, ry, rz], a, v)
    movel(p[x_c + 0.057464, y_c + -0.104542, z_c, rx, ry, rz], a, v)
    movel(p[x_c + 0.057485, y_c + -0.104562, z_c, rx, ry, rz], a, v)
    movel(p[x_c + 0.057507, y_c + -0.104582, z_c, rx, ry, rz], a, v)
    movel(p[x_c + 0.057530, y_c + -0.104603, z_c, rx, ry, rz], a, v)
    movel(p[x_c + 0.057530, y_c + -0.104603, z_c, rx, ry, rz], a, v)
    movel(p[x_c + 0.057553, y_c + -0.104624, z_c, rx, ry, rz], a, v)
    movel(p[x_c + 0.057578, y_c + -0.104646, z_c, rx, ry, rz], a, v)
    movel(p[x_c + 0.057604, y_c + -0.104668, z_c, rx, ry, rz], a, v)
    movel(p[x_c + 0.057631, y_c + -0.104690, z_c, rx, ry, rz], a, v)
    movel(p[x_c + 0.057658, y_c + -0.104713, z_c, rx, ry, rz], a, v)
    movel(p[x_c + 0.057687, y_c + -0.104736, z_c, rx, ry, rz], a, v)
    movel(p[x_c + 0.057717, y_c + -0.104760, z_c, rx, ry, rz], a, v)
    movel(p[x_c + 0.057747, y_c + -0.104784, z_c, rx, ry, rz], a, v)
    movel(p[x_c + 0.057779, y_c + -0.104808, z_c, rx, ry, rz], a, v)
    movel(p[x_c + 0.057811, y_c + -0.104833, z_c, rx, ry, rz], a, v)
    movel(p[x_c + 0.057844, y_c + -0.104857, z_c, rx, ry, rz], a, v)
    movel(p[x_c + 0.057878, y_c + -0.104882, z_c, rx, ry, rz], a, v)
    movel(p[x_c + 0.057913, y_c + -0.104907, z_c, rx, ry, rz], a, v)
    movel(p[x_c + 0.057948, y_c + -0.104933, z_c, rx, ry, rz], a, v)
    movel(p[x_c + 0.057984, y_c + -0.104958, z_c, rx, ry, rz], a, v)
    movel(p[x_c + 0.058021, y_c + -0.104984, z_c, rx, ry, rz], a, v)
    movel(p[x_c + 0.058059, y_c + -0.105010, z_c, rx, ry, rz], a, v)
    movel(p[x_c + 0.058096, y_c + -0.105036, z_c, rx, ry, rz], a, v)
    movel(p[x_c + 0.058135, y_c + -0.105062, z_c, rx, ry, rz], a, v)
    movel(p[x_c + 0.058174, y_c + -0.105088, z_c, rx, ry, rz], a, v)
    movel(p[x_c + 0.058213, y_c + -0.105114, z_c, rx, ry, rz], a, v)
    movel(p[x_c + 0.058253, y_c + -0.105140, z_c, rx, ry, rz], a, v)
    movel(p[x_c + 0.058294, y_c + -0.105166, z_c, rx, ry, rz], a, v)
    movel(p[x_c + 0.058334, y_c + -0.105193, z_c, rx, ry, rz], a, v)
    movel(p[x_c + 0.058375, y_c + -0.105219, z_c, rx, ry, rz], a, v)
    movel(p[x_c + 0.058417, y_c + -0.105245, z_c, rx, ry, rz], a, v)
    movel(p[x_c + 0.058459, y_c + -0.105271, z_c, rx, ry, rz], a, v)
    movel(p[x_c + 0.058500, y_c + -0.105297, z_c, rx, ry, rz], a, v)
    movel(p[x_c + 0.058543, y_c + -0.105322, z_c, rx, ry, rz], a, v)
    movel(p[x_c + 0.058585, y_c + -0.105348, z_c, rx, ry, rz], a, v)
    movel(p[x_c + 0.058627, y_c + -0.105373, z_c, rx, ry, rz], a, v)
    movel(p[x_c + 0.058670, y_c + -0.105399, z_c, rx, ry, rz], a, v)
    movel(p[x_c + 0.058713, y_c + -0.105424, z_c, rx, ry, rz], a, v)
    movel(p[x_c + 0.058756, y_c + -0.105449, z_c, rx, ry, rz], a, v)
    movel(p[x_c + 0.058798, y_c + -0.105473, z_c, rx, ry, rz], a, v)
    movel(p[x_c + 0.058841, y_c + -0.105498, z_c, rx, ry, rz], a, v)
    movel(p[x_c + 0.058884, y_c + -0.105522, z_c, rx, ry, rz], a, v)
    movel(p[x_c + 0.058926, y_c + -0.105545, z_c, rx, ry, rz], a, v)
    movel(p[x_c + 0.058969, y_c + -0.105569, z_c, rx, ry, rz], a, v)
    movel(p[x_c + 0.059011, y_c + -0.105592, z_c, rx, ry, rz], a, v)
    movel(p[x_c + 0.059053, y_c + -0.105614, z_c, rx, ry, rz], a, v)
    movel(p[x_c + 0.059095, y_c + -0.105637, z_c, rx, ry, rz], a, v)
    movel(p[x_c + 0.059137, y_c + -0.105659, z_c, rx, ry, rz], a, v)
    movel(p[x_c + 0.059179, y_c + -0.105680, z_c, rx, ry, rz], a, v)
    movel(p[x_c + 0.059220, y_c + -0.105701, z_c, rx, ry, rz], a, v)
    movel(p[x_c + 0.059261, y_c + -0.105721, z_c, rx, ry, rz], a, v)
    movel(p[x_c + 0.059301, y_c + -0.105741, z_c, rx, ry, rz], a, v)
    movel(p[x_c + 0.059341, y_c + -0.105761, z_c, rx, ry, rz], a, v)
    movel(p[x_c + 0.059381, y_c + -0.105780, z_c, rx, ry, rz], a, v)
    movel(p[x_c + 0.059381, y_c + -0.105780, z_c, rx, ry, rz], a, v)
    movel(p[x_c + 0.059453, y_c + -0.105815, z_c, rx, ry, rz], a, v)
    movel(p[x_c + 0.059532, y_c + -0.105857, z_c, rx, ry, rz], a, v)
    movel(p[x_c + 0.059617, y_c + -0.105904, z_c, rx, ry, rz], a, v)
    movel(p[x_c + 0.059708, y_c + -0.105956, z_c, rx, ry, rz], a, v)
    movel(p[x_c + 0.059805, y_c + -0.106013, z_c, rx, ry, rz], a, v)
    movel(p[x_c + 0.059907, y_c + -0.106075, z_c, rx, ry, rz], a, v)
    movel(p[x_c + 0.060013, y_c + -0.106141, z_c, rx, ry, rz], a, v)
    movel(p[x_c + 0.060125, y_c + -0.106212, z_c, rx, ry, rz], a, v)
    movel(p[x_c + 0.060240, y_c + -0.106287, z_c, rx, ry, rz], a, v)
    movel(p[x_c + 0.060360, y_c + -0.106365, z_c, rx, ry, rz], a, v)
    movel(p[x_c + 0.060483, y_c + -0.106447, z_c, rx, ry, rz], a, v)
    movel(p[x_c + 0.060609, y_c + -0.106532, z_c, rx, ry, rz], a, v)
    movel(p[x_c + 0.060738, y_c + -0.106620, z_c, rx, ry, rz], a, v)
    movel(p[x_c + 0.060869, y_c + -0.106711, z_c, rx, ry, rz], a, v)
    movel(p[x_c + 0.061003, y_c + -0.106805, z_c, rx, ry, rz], a, v)
    movel(p[x_c + 0.061139, y_c + -0.106900, z_c, rx, ry, rz], a, v)
    movel(p[x_c + 0.061277, y_c + -0.106998, z_c, rx, ry, rz], a, v)
    movel(p[x_c + 0.061415, y_c + -0.107097, z_c, rx, ry, rz], a, v)
    movel(p[x_c + 0.061555, y_c + -0.107198, z_c, rx, ry, rz], a, v)
    movel(p[x_c + 0.061695, y_c + -0.107300, z_c, rx, ry, rz], a, v)
    movel(p[x_c + 0.061836, y_c + -0.107404, z_c, rx, ry, rz], a, v)
    movel(p[x_c + 0.061976, y_c + -0.107508, z_c, rx, ry, rz], a, v)
    movel(p[x_c + 0.062116, y_c + -0.107612, z_c, rx, ry, rz], a, v)
    movel(p[x_c + 0.062255, y_c + -0.107717, z_c, rx, ry, rz], a, v)
    movel(p[x_c + 0.062394, y_c + -0.107821, z_c, rx, ry, rz], a, v)
    movel(p[x_c + 0.062530, y_c + -0.107926, z_c, rx, ry, rz], a, v)
    movel(p[x_c + 0.062665, y_c + -0.108029, z_c, rx, ry, rz], a, v)
    movel(p[x_c + 0.062799, y_c + -0.108133, z_c, rx, ry, rz], a, v)
    movel(p[x_c + 0.062929, y_c + -0.108235, z_c, rx, ry, rz], a, v)
    movel(p[x_c + 0.063057, y_c + -0.108336, z_c, rx, ry, rz], a, v)
    movel(p[x_c + 0.063182, y_c + -0.108435, z_c, rx, ry, rz], a, v)
    movel(p[x_c + 0.063304, y_c + -0.108533, z_c, rx, ry, rz], a, v)
    movel(p[x_c + 0.063422, y_c + -0.108628, z_c, rx, ry, rz], a, v)
    movel(p[x_c + 0.063536, y_c + -0.108722, z_c, rx, ry, rz], a, v)
    movel(p[x_c + 0.063645, y_c + -0.108812, z_c, rx, ry, rz], a, v)
    movel(p[x_c + 0.063750, y_c + -0.108901, z_c, rx, ry, rz], a, v)
    movel(p[x_c + 0.063850, y_c + -0.108986, z_c, rx, ry, rz], a, v)
    movel(p[x_c + 0.063944, y_c + -0.109068, z_c, rx, ry, rz], a, v)
    movel(p[x_c + 0.064033, y_c + -0.109146, z_c, rx, ry, rz], a, v)
    movel(p[x_c + 0.064116, y_c + -0.109221, z_c, rx, ry, rz], a, v)
    movel(p[x_c + 0.064192, y_c + -0.109291, z_c, rx, ry, rz], a, v)
    movel(p[x_c + 0.064262, y_c + -0.109358, z_c, rx, ry, rz], a, v)
    movel(p[x_c + 0.064325, y_c + -0.109419, z_c, rx, ry, rz], a, v)
    movel(p[x_c + 0.064380, y_c + -0.109476, z_c, rx, ry, rz], a, v)
    movel(p[x_c + 0.064428, y_c + -0.109529, z_c, rx, ry, rz], a, v)
    movel(p[x_c + 0.064468, y_c + -0.109575, z_c, rx, ry, rz], a, v)
    movel(p[x_c + 0.064499, y_c + -0.109617, z_c, rx, ry, rz], a, v)
    movel(p[x_c + 0.064522, y_c + -0.109652, z_c, rx, ry, rz], a, v)
    movel(p[x_c + 0.064536, y_c + -0.109682, z_c, rx, ry, rz], a, v)
    movel(p[x_c + 0.064536, y_c + -0.109682, z_c, rx, ry, rz], a, v)
    movel(p[x_c + 0.064537, y_c + -0.109693, z_c, rx, ry, rz], a, v)
    movel(p[x_c + 0.064533, y_c + -0.109700, z_c, rx, ry, rz], a, v)
    movel(p[x_c + 0.064523, y_c + -0.109704, z_c, rx, ry, rz], a, v)
    movel(p[x_c + 0.064507, y_c + -0.109704, z_c, rx, ry, rz], a, v)
    movel(p[x_c + 0.064486, y_c + -0.109701, z_c, rx, ry, rz], a, v)
    movel(p[x_c + 0.064459, y_c + -0.109694, z_c, rx, ry, rz], a, v)
    movel(p[x_c + 0.064428, y_c + -0.109685, z_c, rx, ry, rz], a, v)
    movel(p[x_c + 0.064391, y_c + -0.109672, z_c, rx, ry, rz], a, v)
    movel(p[x_c + 0.064350, y_c + -0.109657, z_c, rx, ry, rz], a, v)
    movel(p[x_c + 0.064304, y_c + -0.109638, z_c, rx, ry, rz], a, v)
    movel(p[x_c + 0.064253, y_c + -0.109617, z_c, rx, ry, rz], a, v)
    movel(p[x_c + 0.064198, y_c + -0.109592, z_c, rx, ry, rz], a, v)
    movel(p[x_c + 0.064139, y_c + -0.109566, z_c, rx, ry, rz], a, v)
    movel(p[x_c + 0.064076, y_c + -0.109536, z_c, rx, ry, rz], a, v)
    movel(p[x_c + 0.064008, y_c + -0.109504, z_c, rx, ry, rz], a, v)
    movel(p[x_c + 0.063937, y_c + -0.109470, z_c, rx, ry, rz], a, v)
    movel(p[x_c + 0.063863, y_c + -0.109433, z_c, rx, ry, rz], a, v)
    movel(p[x_c + 0.063785, y_c + -0.109394, z_c, rx, ry, rz], a, v)
    movel(p[x_c + 0.063703, y_c + -0.109352, z_c, rx, ry, rz], a, v)
    movel(p[x_c + 0.063619, y_c + -0.109309, z_c, rx, ry, rz], a, v)
    movel(p[x_c + 0.063531, y_c + -0.109264, z_c, rx, ry, rz], a, v)
    movel(p[x_c + 0.063441, y_c + -0.109216, z_c, rx, ry, rz], a, v)
    movel(p[x_c + 0.063348, y_c + -0.109167, z_c, rx, ry, rz], a, v)
    movel(p[x_c + 0.063252, y_c + -0.109116, z_c, rx, ry, rz], a, v)
    movel(p[x_c + 0.063154, y_c + -0.109063, z_c, rx, ry, rz], a, v)
    movel(p[x_c + 0.063053, y_c + -0.109009, z_c, rx, ry, rz], a, v)
    movel(p[x_c + 0.062951, y_c + -0.108952, z_c, rx, ry, rz], a, v)
    movel(p[x_c + 0.062846, y_c + -0.108895, z_c, rx, ry, rz], a, v)
    movel(p[x_c + 0.062740, y_c + -0.108836, z_c, rx, ry, rz], a, v)
    movel(p[x_c + 0.062632, y_c + -0.108776, z_c, rx, ry, rz], a, v)
    movel(p[x_c + 0.062522, y_c + -0.108715, z_c, rx, ry, rz], a, v)
    movel(p[x_c + 0.062411, y_c + -0.108652, z_c, rx, ry, rz], a, v)
    movel(p[x_c + 0.062299, y_c + -0.108588, z_c, rx, ry, rz], a, v)
    movel(p[x_c + 0.062186, y_c + -0.108524, z_c, rx, ry, rz], a, v)
    movel(p[x_c + 0.062071, y_c + -0.108458, z_c, rx, ry, rz], a, v)
    movel(p[x_c + 0.061957, y_c + -0.108392, z_c, rx, ry, rz], a, v)
    movel(p[x_c + 0.061841, y_c + -0.108324, z_c, rx, ry, rz], a, v)
    movel(p[x_c + 0.061725, y_c + -0.108257, z_c, rx, ry, rz], a, v)
    movel(p[x_c + 0.061608, y_c + -0.108188, z_c, rx, ry, rz], a, v)
    movel(p[x_c + 0.061492, y_c + -0.108119, z_c, rx, ry, rz], a, v)
    movel(p[x_c + 0.061375, y_c + -0.108050, z_c, rx, ry, rz], a, v)
    movel(p[x_c + 0.061259, y_c + -0.107980, z_c, rx, ry, rz], a, v)
    movel(p[x_c + 0.061143, y_c + -0.107910, z_c, rx, ry, rz], a, v)
    movel(p[x_c + 0.061027, y_c + -0.107840, z_c, rx, ry, rz], a, v)
    movel(p[x_c + 0.060912, y_c + -0.107770, z_c, rx, ry, rz], a, v)
    movel(p[x_c + 0.060797, y_c + -0.107700, z_c, rx, ry, rz], a, v)
    movel(p[x_c + 0.060684, y_c + -0.107629, z_c, rx, ry, rz], a, v)
    movel(p[x_c + 0.060571, y_c + -0.107559, z_c, rx, ry, rz], a, v)
    movel(p[x_c + 0.060460, y_c + -0.107489, z_c, rx, ry, rz], a, v)
    movel(p[x_c + 0.060460, y_c + -0.107489, z_c, rx, ry, rz], a, v)
    movel(p[x_c + 0.060350, y_c + -0.107421, z_c, rx, ry, rz], a, v)
    movel(p[x_c + 0.060237, y_c + -0.107351, z_c, rx, ry, rz], a, v)
    movel(p[x_c + 0.060122, y_c + -0.107281, z_c, rx, ry, rz], a, v)
    movel(p[x_c + 0.060004, y_c + -0.107209, z_c, rx, ry, rz], a, v)
    movel(p[x_c + 0.059884, y_c + -0.107137, z_c, rx, ry, rz], a, v)
    movel(p[x_c + 0.059761, y_c + -0.107065, z_c, rx, ry, rz], a, v)
    movel(p[x_c + 0.059637, y_c + -0.106992, z_c, rx, ry, rz], a, v)
    movel(p[x_c + 0.059511, y_c + -0.106918, z_c, rx, ry, rz], a, v)
    movel(p[x_c + 0.059384, y_c + -0.106844, z_c, rx, ry, rz], a, v)
    movel(p[x_c + 0.059255, y_c + -0.106770, z_c, rx, ry, rz], a, v)
    movel(p[x_c + 0.059126, y_c + -0.106697, z_c, rx, ry, rz], a, v)
    movel(p[x_c + 0.058995, y_c + -0.106623, z_c, rx, ry, rz], a, v)
    movel(p[x_c + 0.058865, y_c + -0.106549, z_c, rx, ry, rz], a, v)
    movel(p[x_c + 0.058733, y_c + -0.106476, z_c, rx, ry, rz], a, v)
    movel(p[x_c + 0.058602, y_c + -0.106403, z_c, rx, ry, rz], a, v)
    movel(p[x_c + 0.058471, y_c + -0.106331, z_c, rx, ry, rz], a, v)
    movel(p[x_c + 0.058340, y_c + -0.106259, z_c, rx, ry, rz], a, v)
    movel(p[x_c + 0.058209, y_c + -0.106188, z_c, rx, ry, rz], a, v)
    movel(p[x_c + 0.058080, y_c + -0.106118, z_c, rx, ry, rz], a, v)
    movel(p[x_c + 0.057951, y_c + -0.106050, z_c, rx, ry, rz], a, v)
    movel(p[x_c + 0.057824, y_c + -0.105982, z_c, rx, ry, rz], a, v)
    movel(p[x_c + 0.057698, y_c + -0.105915, z_c, rx, ry, rz], a, v)
    movel(p[x_c + 0.057573, y_c + -0.105850, z_c, rx, ry, rz], a, v)
    movel(p[x_c + 0.057451, y_c + -0.105786, z_c, rx, ry, rz], a, v)
    movel(p[x_c + 0.057330, y_c + -0.105724, z_c, rx, ry, rz], a, v)
    movel(p[x_c + 0.057212, y_c + -0.105663, z_c, rx, ry, rz], a, v)
    movel(p[x_c + 0.057097, y_c + -0.105605, z_c, rx, ry, rz], a, v)
    movel(p[x_c + 0.056984, y_c + -0.105548, z_c, rx, ry, rz], a, v)
    movel(p[x_c + 0.056874, y_c + -0.105493, z_c, rx, ry, rz], a, v)
    movel(p[x_c + 0.056768, y_c + -0.105441, z_c, rx, ry, rz], a, v)
    movel(p[x_c + 0.056665, y_c + -0.105390, z_c, rx, ry, rz], a, v)
    movel(p[x_c + 0.056565, y_c + -0.105343, z_c, rx, ry, rz], a, v)
    movel(p[x_c + 0.056469, y_c + -0.105297, z_c, rx, ry, rz], a, v)
    movel(p[x_c + 0.056378, y_c + -0.105254, z_c, rx, ry, rz], a, v)
    movel(p[x_c + 0.056291, y_c + -0.105214, z_c, rx, ry, rz], a, v)
    movel(p[x_c + 0.056208, y_c + -0.105177, z_c, rx, ry, rz], a, v)
    movel(p[x_c + 0.056130, y_c + -0.105143, z_c, rx, ry, rz], a, v)
    movel(p[x_c + 0.056057, y_c + -0.105111, z_c, rx, ry, rz], a, v)
    movel(p[x_c + 0.055989, y_c + -0.105083, z_c, rx, ry, rz], a, v)
    movel(p[x_c + 0.055927, y_c + -0.105059, z_c, rx, ry, rz], a, v)
    movel(p[x_c + 0.055870, y_c + -0.105037, z_c, rx, ry, rz], a, v)
    movel(p[x_c + 0.055819, y_c + -0.105019, z_c, rx, ry, rz], a, v)
    movel(p[x_c + 0.055774, y_c + -0.105005, z_c, rx, ry, rz], a, v)
    movel(p[x_c + 0.055735, y_c + -0.104995, z_c, rx, ry, rz], a, v)
    movel(p[x_c + 0.055703, y_c + -0.104988, z_c, rx, ry, rz], a, v)
    movel(p[x_c + 0.055678, y_c + -0.104985, z_c, rx, ry, rz], a, v)
    movel(p[x_c + 0.055660, y_c + -0.104987, z_c, rx, ry, rz], a, v)
    movel(p[x_c + 0.055649, y_c + -0.104993, z_c, rx, ry, rz], a, v)
    movel(p[x_c + 0.055645, y_c + -0.105003, z_c, rx, ry, rz], a, v)
    movel(p[x_c + 0.055645, y_c + -0.105003, z_c, rx, ry, rz], a, v)
    movel(p[x_c + 0.055645, y_c + -0.105010, z_c, rx, ry, rz], a, v)
    movel(p[x_c + 0.055645, y_c + -0.105016, z_c, rx, ry, rz], a, v)
    movel(p[x_c + 0.055646, y_c + -0.105023, z_c, rx, ry, rz], a, v)
    movel(p[x_c + 0.055646, y_c + -0.105030, z_c, rx, ry, rz], a, v)
    movel(p[x_c + 0.055647, y_c + -0.105037, z_c, rx, ry, rz], a, v)
    movel(p[x_c + 0.055648, y_c + -0.105043, z_c, rx, ry, rz], a, v)
    movel(p[x_c + 0.055649, y_c + -0.105050, z_c, rx, ry, rz], a, v)
    movel(p[x_c + 0.055651, y_c + -0.105056, z_c, rx, ry, rz], a, v)
    movel(p[x_c + 0.055652, y_c + -0.105062, z_c, rx, ry, rz], a, v)
    movel(p[x_c + 0.055654, y_c + -0.105069, z_c, rx, ry, rz], a, v)
    movel(p[x_c + 0.055655, y_c + -0.105075, z_c, rx, ry, rz], a, v)
    movel(p[x_c + 0.055657, y_c + -0.105081, z_c, rx, ry, rz], a, v)
    movel(p[x_c + 0.055660, y_c + -0.105087, z_c, rx, ry, rz], a, v)
    movel(p[x_c + 0.055662, y_c + -0.105093, z_c, rx, ry, rz], a, v)
    movel(p[x_c + 0.055664, y_c + -0.105099, z_c, rx, ry, rz], a, v)
    movel(p[x_c + 0.055667, y_c + -0.105104, z_c, rx, ry, rz], a, v)
    movel(p[x_c + 0.055669, y_c + -0.105110, z_c, rx, ry, rz], a, v)
    movel(p[x_c + 0.055672, y_c + -0.105115, z_c, rx, ry, rz], a, v)
    movel(p[x_c + 0.055675, y_c + -0.105121, z_c, rx, ry, rz], a, v)
    movel(p[x_c + 0.055678, y_c + -0.105126, z_c, rx, ry, rz], a, v)
    movel(p[x_c + 0.055682, y_c + -0.105131, z_c, rx, ry, rz], a, v)
    movel(p[x_c + 0.055685, y_c + -0.105136, z_c, rx, ry, rz], a, v)
    movel(p[x_c + 0.055688, y_c + -0.105141, z_c, rx, ry, rz], a, v)
    movel(p[x_c + 0.055692, y_c + -0.105146, z_c, rx, ry, rz], a, v)
    movel(p[x_c + 0.055696, y_c + -0.105150, z_c, rx, ry, rz], a, v)
    movel(p[x_c + 0.055700, y_c + -0.105155, z_c, rx, ry, rz], a, v)
    movel(p[x_c + 0.055704, y_c + -0.105159, z_c, rx, ry, rz], a, v)
    movel(p[x_c + 0.055708, y_c + -0.105163, z_c, rx, ry, rz], a, v)
    movel(p[x_c + 0.055712, y_c + -0.105167, z_c, rx, ry, rz], a, v)
    movel(p[x_c + 0.055716, y_c + -0.105171, z_c, rx, ry, rz], a, v)
    movel(p[x_c + 0.055720, y_c + -0.105175, z_c, rx, ry, rz], a, v)
    movel(p[x_c + 0.055725, y_c + -0.105178, z_c, rx, ry, rz], a, v)
    movel(p[x_c + 0.055729, y_c + -0.105181, z_c, rx, ry, rz], a, v)
    movel(p[x_c + 0.055734, y_c + -0.105185, z_c, rx, ry, rz], a, v)
    movel(p[x_c + 0.055739, y_c + -0.105188, z_c, rx, ry, rz], a, v)
    movel(p[x_c + 0.055743, y_c + -0.105190, z_c, rx, ry, rz], a, v)
    movel(p[x_c + 0.055748, y_c + -0.105193, z_c, rx, ry, rz], a, v)
    movel(p[x_c + 0.055753, y_c + -0.105195, z_c, rx, ry, rz], a, v)
    movel(p[x_c + 0.055758, y_c + -0.105198, z_c, rx, ry, rz], a, v)
    movel(p[x_c + 0.055763, y_c + -0.105200, z_c, rx, ry, rz], a, v)
    movel(p[x_c + 0.055768, y_c + -0.105202, z_c, rx, ry, rz], a, v)
    movel(p[x_c + 0.055774, y_c + -0.105203, z_c, rx, ry, rz], a, v)
    movel(p[x_c + 0.055779, y_c + -0.105205, z_c, rx, ry, rz], a, v)
    movel(p[x_c + 0.055784, y_c + -0.105206, z_c, rx, ry, rz], a, v)
    movel(p[x_c + 0.055790, y_c + -0.105207, z_c, rx, ry, rz], a, v)
    movel(p[x_c + 0.055795, y_c + -0.105208, z_c, rx, ry, rz], a, v)
    movel(p[x_c + 0.055801, y_c + -0.105208, z_c, rx, ry, rz], a, v)
    movel(p[x_c + 0.055806, y_c + -0.105209, z_c, rx, ry, rz], a, v)
    movel(p[x_c + 0.055812, y_c + -0.105209, z_c, rx, ry, rz], a, v)
    movel(p[x_c + 0.055812, y_c + -0.105209, z_c, rx, ry, rz], a, v)
    movel(p[x_c + 0.055825, y_c + -0.105213, z_c, rx, ry, rz], a, v)
    movel(p[x_c + 0.055847, y_c + -0.105225, z_c, rx, ry, rz], a, v)
    movel(p[x_c + 0.055878, y_c + -0.105244, z_c, rx, ry, rz], a, v)
    movel(p[x_c + 0.055917, y_c + -0.105271, z_c, rx, ry, rz], a, v)
    movel(p[x_c + 0.055965, y_c + -0.105305, z_c, rx, ry, rz], a, v)
    movel(p[x_c + 0.056020, y_c + -0.105345, z_c, rx, ry, rz], a, v)
    movel(p[x_c + 0.056082, y_c + -0.105392, z_c, rx, ry, rz], a, v)
    movel(p[x_c + 0.056152, y_c + -0.105445, z_c, rx, ry, rz], a, v)
    movel(p[x_c + 0.056227, y_c + -0.105503, z_c, rx, ry, rz], a, v)
    movel(p[x_c + 0.056310, y_c + -0.105567, z_c, rx, ry, rz], a, v)
    movel(p[x_c + 0.056397, y_c + -0.105636, z_c, rx, ry, rz], a, v)
    movel(p[x_c + 0.056491, y_c + -0.105710, z_c, rx, ry, rz], a, v)
    movel(p[x_c + 0.056589, y_c + -0.105788, z_c, rx, ry, rz], a, v)
    movel(p[x_c + 0.056692, y_c + -0.105870, z_c, rx, ry, rz], a, v)
    movel(p[x_c + 0.056800, y_c + -0.105956, z_c, rx, ry, rz], a, v)
    movel(p[x_c + 0.056911, y_c + -0.106046, z_c, rx, ry, rz], a, v)
    movel(p[x_c + 0.057026, y_c + -0.106139, z_c, rx, ry, rz], a, v)
    movel(p[x_c + 0.057144, y_c + -0.106235, z_c, rx, ry, rz], a, v)
    movel(p[x_c + 0.057265, y_c + -0.106333, z_c, rx, ry, rz], a, v)
    movel(p[x_c + 0.057388, y_c + -0.106434, z_c, rx, ry, rz], a, v)
    movel(p[x_c + 0.057514, y_c + -0.106537, z_c, rx, ry, rz], a, v)
    movel(p[x_c + 0.057641, y_c + -0.106641, z_c, rx, ry, rz], a, v)
    movel(p[x_c + 0.057769, y_c + -0.106747, z_c, rx, ry, rz], a, v)
    movel(p[x_c + 0.057898, y_c + -0.106854, z_c, rx, ry, rz], a, v)
    movel(p[x_c + 0.058028, y_c + -0.106961, z_c, rx, ry, rz], a, v)
    movel(p[x_c + 0.058158, y_c + -0.107069, z_c, rx, ry, rz], a, v)
    movel(p[x_c + 0.058288, y_c + -0.107177, z_c, rx, ry, rz], a, v)
    movel(p[x_c + 0.058417, y_c + -0.107285, z_c, rx, ry, rz], a, v)
    movel(p[x_c + 0.058545, y_c + -0.107393, z_c, rx, ry, rz], a, v)
    movel(p[x_c + 0.058672, y_c + -0.107499, z_c, rx, ry, rz], a, v)
    movel(p[x_c + 0.058797, y_c + -0.107605, z_c, rx, ry, rz], a, v)
    movel(p[x_c + 0.058920, y_c + -0.107708, z_c, rx, ry, rz], a, v)
    movel(p[x_c + 0.059041, y_c + -0.107811, z_c, rx, ry, rz], a, v)
    movel(p[x_c + 0.059159, y_c + -0.107911, z_c, rx, ry, rz], a, v)
    movel(p[x_c + 0.059274, y_c + -0.108009, z_c, rx, ry, rz], a, v)
    movel(p[x_c + 0.059385, y_c + -0.108104, z_c, rx, ry, rz], a, v)
    movel(p[x_c + 0.059492, y_c + -0.108196, z_c, rx, ry, rz], a, v)
    movel(p[x_c + 0.059595, y_c + -0.108284, z_c, rx, ry, rz], a, v)
    movel(p[x_c + 0.059693, y_c + -0.108370, z_c, rx, ry, rz], a, v)
    movel(p[x_c + 0.059786, y_c + -0.108451, z_c, rx, ry, rz], a, v)
    movel(p[x_c + 0.059873, y_c + -0.108528, z_c, rx, ry, rz], a, v)
    movel(p[x_c + 0.059955, y_c + -0.108600, z_c, rx, ry, rz], a, v)
    movel(p[x_c + 0.060031, y_c + -0.108668, z_c, rx, ry, rz], a, v)
    movel(p[x_c + 0.060100, y_c + -0.108730, z_c, rx, ry, rz], a, v)
    movel(p[x_c + 0.060162, y_c + -0.108787, z_c, rx, ry, rz], a, v)
    movel(p[x_c + 0.060216, y_c + -0.108838, z_c, rx, ry, rz], a, v)
    movel(p[x_c + 0.060263, y_c + -0.108883, z_c, rx, ry, rz], a, v)
    movel(p[x_c + 0.060302, y_c + -0.108921, z_c, rx, ry, rz], a, v)
    movel(p[x_c + 0.060332, y_c + -0.108953, z_c, rx, ry, rz], a, v)
    movel(p[x_c + 0.060332, y_c + -0.108953, z_c, rx, ry, rz], a, v)
    movel(p[x_c + 0.060342, y_c + -0.108963, z_c, rx, ry, rz], a, v)
    movel(p[x_c + 0.060349, y_c + -0.108972, z_c, rx, ry, rz], a, v)
    movel(p[x_c + 0.060355, y_c + -0.108980, z_c, rx, ry, rz], a, v)
    movel(p[x_c + 0.060358, y_c + -0.108987, z_c, rx, ry, rz], a, v)
    movel(p[x_c + 0.060360, y_c + -0.108992, z_c, rx, ry, rz], a, v)
    movel(p[x_c + 0.060360, y_c + -0.108996, z_c, rx, ry, rz], a, v)
    movel(p[x_c + 0.060358, y_c + -0.108998, z_c, rx, ry, rz], a, v)
    movel(p[x_c + 0.060355, y_c + -0.109000, z_c, rx, ry, rz], a, v)
    movel(p[x_c + 0.060349, y_c + -0.108999, z_c, rx, ry, rz], a, v)
    movel(p[x_c + 0.060341, y_c + -0.108998, z_c, rx, ry, rz], a, v)
    movel(p[x_c + 0.060331, y_c + -0.108995, z_c, rx, ry, rz], a, v)
    movel(p[x_c + 0.060320, y_c + -0.108990, z_c, rx, ry, rz], a, v)
    movel(p[x_c + 0.060306, y_c + -0.108985, z_c, rx, ry, rz], a, v)
    movel(p[x_c + 0.060290, y_c + -0.108977, z_c, rx, ry, rz], a, v)
    movel(p[x_c + 0.060272, y_c + -0.108969, z_c, rx, ry, rz], a, v)
    movel(p[x_c + 0.060251, y_c + -0.108959, z_c, rx, ry, rz], a, v)
    movel(p[x_c + 0.060229, y_c + -0.108947, z_c, rx, ry, rz], a, v)
    movel(p[x_c + 0.060204, y_c + -0.108934, z_c, rx, ry, rz], a, v)
    movel(p[x_c + 0.060178, y_c + -0.108919, z_c, rx, ry, rz], a, v)
    movel(p[x_c + 0.060149, y_c + -0.108903, z_c, rx, ry, rz], a, v)
    movel(p[x_c + 0.060117, y_c + -0.108885, z_c, rx, ry, rz], a, v)
    movel(p[x_c + 0.060084, y_c + -0.108866, z_c, rx, ry, rz], a, v)
    movel(p[x_c + 0.060048, y_c + -0.108845, z_c, rx, ry, rz], a, v)
    movel(p[x_c + 0.060010, y_c + -0.108823, z_c, rx, ry, rz], a, v)
    movel(p[x_c + 0.059969, y_c + -0.108798, z_c, rx, ry, rz], a, v)
    movel(p[x_c + 0.059926, y_c + -0.108773, z_c, rx, ry, rz], a, v)
    movel(p[x_c + 0.059880, y_c + -0.108745, z_c, rx, ry, rz], a, v)
    movel(p[x_c + 0.059832, y_c + -0.108716, z_c, rx, ry, rz], a, v)
    movel(p[x_c + 0.059782, y_c + -0.108686, z_c, rx, ry, rz], a, v)
    movel(p[x_c + 0.059729, y_c + -0.108653, z_c, rx, ry, rz], a, v)
    movel(p[x_c + 0.059674, y_c + -0.108619, z_c, rx, ry, rz], a, v)
    movel(p[x_c + 0.059616, y_c + -0.108583, z_c, rx, ry, rz], a, v)
    movel(p[x_c + 0.059555, y_c + -0.108546, z_c, rx, ry, rz], a, v)
    movel(p[x_c + 0.059492, y_c + -0.108506, z_c, rx, ry, rz], a, v)
    movel(p[x_c + 0.059426, y_c + -0.108465, z_c, rx, ry, rz], a, v)
    movel(p[x_c + 0.059357, y_c + -0.108422, z_c, rx, ry, rz], a, v)
    movel(p[x_c + 0.059286, y_c + -0.108378, z_c, rx, ry, rz], a, v)
    movel(p[x_c + 0.059212, y_c + -0.108331, z_c, rx, ry, rz], a, v)
    movel(p[x_c + 0.059136, y_c + -0.108283, z_c, rx, ry, rz], a, v)
    movel(p[x_c + 0.059056, y_c + -0.108233, z_c, rx, ry, rz], a, v)
    movel(p[x_c + 0.058974, y_c + -0.108181, z_c, rx, ry, rz], a, v)
    movel(p[x_c + 0.058889, y_c + -0.108127, z_c, rx, ry, rz], a, v)
    movel(p[x_c + 0.058801, y_c + -0.108071, z_c, rx, ry, rz], a, v)
    movel(p[x_c + 0.058710, y_c + -0.108013, z_c, rx, ry, rz], a, v)
    movel(p[x_c + 0.058616, y_c + -0.107954, z_c, rx, ry, rz], a, v)
    movel(p[x_c + 0.058520, y_c + -0.107892, z_c, rx, ry, rz], a, v)
    movel(p[x_c + 0.058420, y_c + -0.107829, z_c, rx, ry, rz], a, v)
    movel(p[x_c + 0.058318, y_c + -0.107763, z_c, rx, ry, rz], a, v)
    movel(p[x_c + 0.058212, y_c + -0.107696, z_c, rx, ry, rz], a, v)
    movel(p[x_c + 0.058212, y_c + -0.107696, z_c, rx, ry, rz], a, v)
    movel(p[x_c + 0.058013, y_c + -0.107569, z_c, rx, ry, rz], a, v)
    movel(p[x_c + 0.057814, y_c + -0.107442, z_c, rx, ry, rz], a, v)
    movel(p[x_c + 0.057616, y_c + -0.107316, z_c, rx, ry, rz], a, v)
    movel(p[x_c + 0.057417, y_c + -0.107191, z_c, rx, ry, rz], a, v)
    movel(p[x_c + 0.057218, y_c + -0.107066, z_c, rx, ry, rz], a, v)
    movel(p[x_c + 0.057020, y_c + -0.106942, z_c, rx, ry, rz], a, v)
    movel(p[x_c + 0.056823, y_c + -0.106818, z_c, rx, ry, rz], a, v)
    movel(p[x_c + 0.056627, y_c + -0.106696, z_c, rx, ry, rz], a, v)
    movel(p[x_c + 0.056432, y_c + -0.106575, z_c, rx, ry, rz], a, v)
    movel(p[x_c + 0.056238, y_c + -0.106454, z_c, rx, ry, rz], a, v)
    movel(p[x_c + 0.056046, y_c + -0.106336, z_c, rx, ry, rz], a, v)
    movel(p[x_c + 0.055855, y_c + -0.106218, z_c, rx, ry, rz], a, v)
    movel(p[x_c + 0.055666, y_c + -0.106103, z_c, rx, ry, rz], a, v)
    movel(p[x_c + 0.055480, y_c + -0.105989, z_c, rx, ry, rz], a, v)
    movel(p[x_c + 0.055296, y_c + -0.105876, z_c, rx, ry, rz], a, v)
    movel(p[x_c + 0.055114, y_c + -0.105766, z_c, rx, ry, rz], a, v)
    movel(p[x_c + 0.054935, y_c + -0.105657, z_c, rx, ry, rz], a, v)
    movel(p[x_c + 0.054759, y_c + -0.105551, z_c, rx, ry, rz], a, v)
    movel(p[x_c + 0.054586, y_c + -0.105447, z_c, rx, ry, rz], a, v)
    movel(p[x_c + 0.054416, y_c + -0.105346, z_c, rx, ry, rz], a, v)
    movel(p[x_c + 0.054250, y_c + -0.105246, z_c, rx, ry, rz], a, v)
    movel(p[x_c + 0.054088, y_c + -0.105150, z_c, rx, ry, rz], a, v)
    movel(p[x_c + 0.053929, y_c + -0.105056, z_c, rx, ry, rz], a, v)
    movel(p[x_c + 0.053775, y_c + -0.104965, z_c, rx, ry, rz], a, v)
    movel(p[x_c + 0.053625, y_c + -0.104877, z_c, rx, ry, rz], a, v)
    movel(p[x_c + 0.053479, y_c + -0.104792, z_c, rx, ry, rz], a, v)
    movel(p[x_c + 0.053338, y_c + -0.104710, z_c, rx, ry, rz], a, v)
    movel(p[x_c + 0.053202, y_c + -0.104632, z_c, rx, ry, rz], a, v)
    movel(p[x_c + 0.053071, y_c + -0.104557, z_c, rx, ry, rz], a, v)
    movel(p[x_c + 0.052945, y_c + -0.104485, z_c, rx, ry, rz], a, v)
    movel(p[x_c + 0.052825, y_c + -0.104417, z_c, rx, ry, rz], a, v)
    movel(p[x_c + 0.052711, y_c + -0.104353, z_c, rx, ry, rz], a, v)
    movel(p[x_c + 0.052602, y_c + -0.104293, z_c, rx, ry, rz], a, v)
    movel(p[x_c + 0.052499, y_c + -0.104237, z_c, rx, ry, rz], a, v)
    movel(p[x_c + 0.052403, y_c + -0.104185, z_c, rx, ry, rz], a, v)
    movel(p[x_c + 0.052313, y_c + -0.104137, z_c, rx, ry, rz], a, v)
    movel(p[x_c + 0.052230, y_c + -0.104093, z_c, rx, ry, rz], a, v)
    movel(p[x_c + 0.052154, y_c + -0.104054, z_c, rx, ry, rz], a, v)
    movel(p[x_c + 0.052085, y_c + -0.104020, z_c, rx, ry, rz], a, v)
    movel(p[x_c + 0.052023, y_c + -0.103990, z_c, rx, ry, rz], a, v)
    movel(p[x_c + 0.051969, y_c + -0.103965, z_c, rx, ry, rz], a, v)
    movel(p[x_c + 0.051922, y_c + -0.103945, z_c, rx, ry, rz], a, v)
    movel(p[x_c + 0.051883, y_c + -0.103930, z_c, rx, ry, rz], a, v)
    movel(p[x_c + 0.051852, y_c + -0.103920, z_c, rx, ry, rz], a, v)
    movel(p[x_c + 0.051830, y_c + -0.103915, z_c, rx, ry, rz], a, v)
    movel(p[x_c + 0.051815, y_c + -0.103916, z_c, rx, ry, rz], a, v)
    movel(p[x_c + 0.051810, y_c + -0.103922, z_c, rx, ry, rz], a, v)
    movel(p[x_c + 0.051813, y_c + -0.103934, z_c, rx, ry, rz], a, v)
    movel(p[x_c + 0.051826, y_c + -0.103952, z_c, rx, ry, rz], a, v)
    movel(p[x_c + 0.051826, y_c + -0.103952, z_c, rx, ry, rz], a, v)
    movel(p[x_c + 0.051837, y_c + -0.103964, z_c, rx, ry, rz], a, v)
    movel(p[x_c + 0.051849, y_c + -0.103978, z_c, rx, ry, rz], a, v)
    movel(p[x_c + 0.051863, y_c + -0.103993, z_c, rx, ry, rz], a, v)
    movel(p[x_c + 0.051879, y_c + -0.104009, z_c, rx, ry, rz], a, v)
    movel(p[x_c + 0.051896, y_c + -0.104026, z_c, rx, ry, rz], a, v)
    movel(p[x_c + 0.051915, y_c + -0.104045, z_c, rx, ry, rz], a, v)
    movel(p[x_c + 0.051936, y_c + -0.104065, z_c, rx, ry, rz], a, v)
    movel(p[x_c + 0.051958, y_c + -0.104086, z_c, rx, ry, rz], a, v)
    movel(p[x_c + 0.051982, y_c + -0.104108, z_c, rx, ry, rz], a, v)
    movel(p[x_c + 0.052007, y_c + -0.104131, z_c, rx, ry, rz], a, v)
    movel(p[x_c + 0.052034, y_c + -0.104155, z_c, rx, ry, rz], a, v)
    movel(p[x_c + 0.052062, y_c + -0.104180, z_c, rx, ry, rz], a, v)
    movel(p[x_c + 0.052091, y_c + -0.104207, z_c, rx, ry, rz], a, v)
    movel(p[x_c + 0.052122, y_c + -0.104234, z_c, rx, ry, rz], a, v)
    movel(p[x_c + 0.052154, y_c + -0.104262, z_c, rx, ry, rz], a, v)
    movel(p[x_c + 0.052187, y_c + -0.104291, z_c, rx, ry, rz], a, v)
    movel(p[x_c + 0.052221, y_c + -0.104321, z_c, rx, ry, rz], a, v)
    movel(p[x_c + 0.052257, y_c + -0.104351, z_c, rx, ry, rz], a, v)
    movel(p[x_c + 0.052294, y_c + -0.104383, z_c, rx, ry, rz], a, v)
    movel(p[x_c + 0.052332, y_c + -0.104415, z_c, rx, ry, rz], a, v)
    movel(p[x_c + 0.052371, y_c + -0.104448, z_c, rx, ry, rz], a, v)
    movel(p[x_c + 0.052411, y_c + -0.104482, z_c, rx, ry, rz], a, v)
    movel(p[x_c + 0.052452, y_c + -0.104517, z_c, rx, ry, rz], a, v)
    movel(p[x_c + 0.052495, y_c + -0.104552, z_c, rx, ry, rz], a, v)
    movel(p[x_c + 0.052538, y_c + -0.104588, z_c, rx, ry, rz], a, v)
    movel(p[x_c + 0.052582, y_c + -0.104624, z_c, rx, ry, rz], a, v)
    movel(p[x_c + 0.052627, y_c + -0.104661, z_c, rx, ry, rz], a, v)
    movel(p[x_c + 0.052672, y_c + -0.104699, z_c, rx, ry, rz], a, v)
    movel(p[x_c + 0.052719, y_c + -0.104737, z_c, rx, ry, rz], a, v)
    movel(p[x_c + 0.052766, y_c + -0.104775, z_c, rx, ry, rz], a, v)
    movel(p[x_c + 0.052814, y_c + -0.104815, z_c, rx, ry, rz], a, v)
    movel(p[x_c + 0.052863, y_c + -0.104854, z_c, rx, ry, rz], a, v)
    movel(p[x_c + 0.052913, y_c + -0.104894, z_c, rx, ry, rz], a, v)
    movel(p[x_c + 0.052963, y_c + -0.104934, z_c, rx, ry, rz], a, v)
    movel(p[x_c + 0.053013, y_c + -0.104975, z_c, rx, ry, rz], a, v)
    movel(p[x_c + 0.053065, y_c + -0.105016, z_c, rx, ry, rz], a, v)
    movel(p[x_c + 0.053117, y_c + -0.105058, z_c, rx, ry, rz], a, v)
    movel(p[x_c + 0.053169, y_c + -0.105099, z_c, rx, ry, rz], a, v)
    movel(p[x_c + 0.053222, y_c + -0.105141, z_c, rx, ry, rz], a, v)
    movel(p[x_c + 0.053275, y_c + -0.105183, z_c, rx, ry, rz], a, v)
    movel(p[x_c + 0.053329, y_c + -0.105225, z_c, rx, ry, rz], a, v)
    movel(p[x_c + 0.053383, y_c + -0.105268, z_c, rx, ry, rz], a, v)
    movel(p[x_c + 0.053437, y_c + -0.105310, z_c, rx, ry, rz], a, v)
    movel(p[x_c + 0.053492, y_c + -0.105353, z_c, rx, ry, rz], a, v)
    movel(p[x_c + 0.053546, y_c + -0.105396, z_c, rx, ry, rz], a, v)
    movel(p[x_c + 0.053602, y_c + -0.105438, z_c, rx, ry, rz], a, v)
    movel(p[x_c + 0.053657, y_c + -0.105481, z_c, rx, ry, rz], a, v)
    movel(p[x_c + 0.053712, y_c + -0.105524, z_c, rx, ry, rz], a, v)
    movel(p[x_c + 0.053768, y_c + -0.105566, z_c, rx, ry, rz], a, v)
    movel(p[x_c + 0.053768, y_c + -0.105566, z_c, rx, ry, rz], a, v)
    movel(p[x_c + 0.053874, y_c + -0.105648, z_c, rx, ry, rz], a, v)
    movel(p[x_c + 0.053976, y_c + -0.105727, z_c, rx, ry, rz], a, v)
    movel(p[x_c + 0.054075, y_c + -0.105803, z_c, rx, ry, rz], a, v)
    movel(p[x_c + 0.054170, y_c + -0.105877, z_c, rx, ry, rz], a, v)
    movel(p[x_c + 0.054262, y_c + -0.105949, z_c, rx, ry, rz], a, v)
    movel(p[x_c + 0.054351, y_c + -0.106018, z_c, rx, ry, rz], a, v)
    movel(p[x_c + 0.054435, y_c + -0.106085, z_c, rx, ry, rz], a, v)
    movel(p[x_c + 0.054516, y_c + -0.106149, z_c, rx, ry, rz], a, v)
    movel(p[x_c + 0.054594, y_c + -0.106211, z_c, rx, ry, rz], a, v)
    movel(p[x_c + 0.054668, y_c + -0.106271, z_c, rx, ry, rz], a, v)
    movel(p[x_c + 0.054739, y_c + -0.106328, z_c, rx, ry, rz], a, v)
    movel(p[x_c + 0.054806, y_c + -0.106383, z_c, rx, ry, rz], a, v)
    movel(p[x_c + 0.054869, y_c + -0.106435, z_c, rx, ry, rz], a, v)
    movel(p[x_c + 0.054929, y_c + -0.106484, z_c, rx, ry, rz], a, v)
    movel(p[x_c + 0.054985, y_c + -0.106532, z_c, rx, ry, rz], a, v)
    movel(p[x_c + 0.055037, y_c + -0.106576, z_c, rx, ry, rz], a, v)
    movel(p[x_c + 0.055086, y_c + -0.106618, z_c, rx, ry, rz], a, v)
    movel(p[x_c + 0.055132, y_c + -0.106658, z_c, rx, ry, rz], a, v)
    movel(p[x_c + 0.055173, y_c + -0.106695, z_c, rx, ry, rz], a, v)
    movel(p[x_c + 0.055211, y_c + -0.106730, z_c, rx, ry, rz], a, v)
    movel(p[x_c + 0.055246, y_c + -0.106762, z_c, rx, ry, rz], a, v)
    movel(p[x_c + 0.055277, y_c + -0.106791, z_c, rx, ry, rz], a, v)
    movel(p[x_c + 0.055304, y_c + -0.106818, z_c, rx, ry, rz], a, v)
    movel(p[x_c + 0.055327, y_c + -0.106843, z_c, rx, ry, rz], a, v)
    movel(p[x_c + 0.055347, y_c + -0.106864, z_c, rx, ry, rz], a, v)
    movel(p[x_c + 0.055363, y_c + -0.106884, z_c, rx, ry, rz], a, v)
    movel(p[x_c + 0.055375, y_c + -0.106900, z_c, rx, ry, rz], a, v)
    movel(p[x_c + 0.055384, y_c + -0.106914, z_c, rx, ry, rz], a, v)
    movel(p[x_c + 0.055389, y_c + -0.106926, z_c, rx, ry, rz], a, v)
    movel(p[x_c + 0.055390, y_c + -0.106934, z_c, rx, ry, rz], a, v)
    movel(p[x_c + 0.055387, y_c + -0.106941, z_c, rx, ry, rz], a, v)
    movel(p[x_c + 0.055381, y_c + -0.106944, z_c, rx, ry, rz], a, v)
    movel(p[x_c + 0.055371, y_c + -0.106945, z_c, rx, ry, rz], a, v)
    movel(p[x_c + 0.055357, y_c + -0.106943, z_c, rx, ry, rz], a, v)
    movel(p[x_c + 0.055340, y_c + -0.106939, z_c, rx, ry, rz], a, v)
    movel(p[x_c + 0.055318, y_c + -0.106932, z_c, rx, ry, rz], a, v)
    movel(p[x_c + 0.055293, y_c + -0.106922, z_c, rx, ry, rz], a, v)
